# B&R Automation Studio project mvDemoTrak
Automation Studio 4.12.4.107 SP; technology packages: mapp 5.22.1, mappCockpit 5.22.0, mappMotion 5.22.1, mappView 5.22.1

## Configuration CP3686X

### Hardware
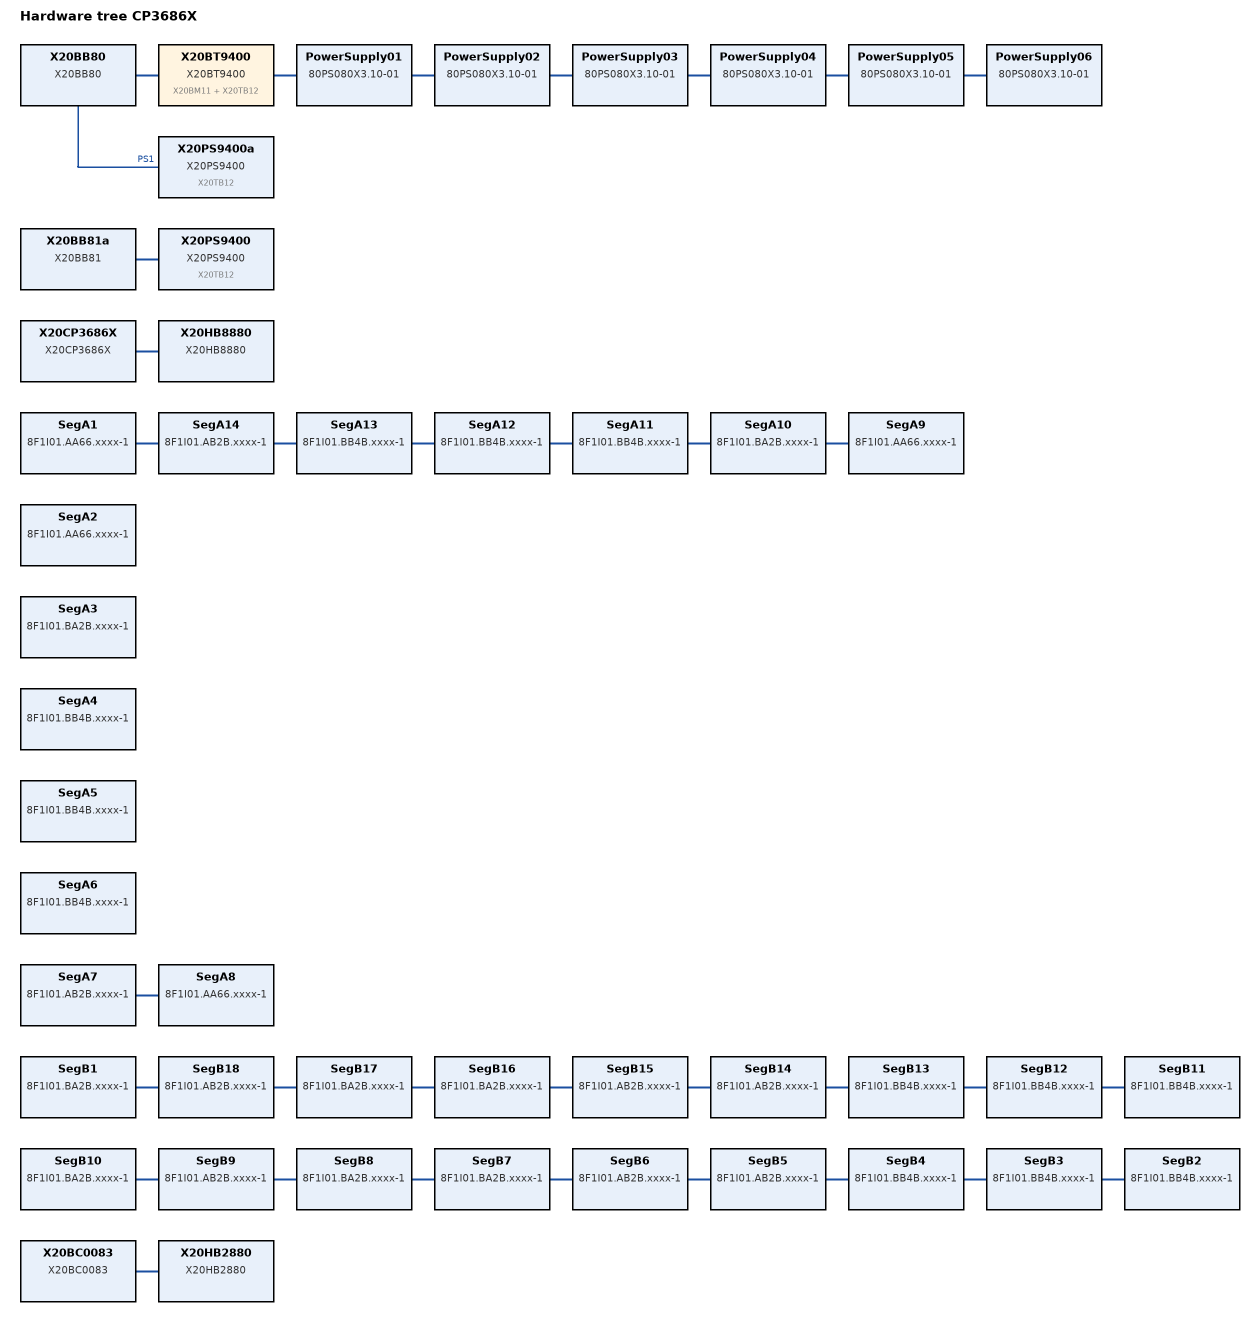
```
PowerSupply01 : 80PS080X3.10-01 v1.5.0.0  [X2X1 -> X20BT9400.X2X1 [Cable Type=X2XCable, Length=10, Version=1.0.0.3]]
  Supervision = off
PowerSupply02 : 80PS080X3.10-01 v1.5.0.0  [X2X1 -> PowerSupply01.X2X2 [Cable Type=X2XCable, Length=10, Version=1.0.0.3]]
  Supervision = off
PowerSupply03 : 80PS080X3.10-01 v1.5.0.0  [X2X1 -> PowerSupply02.X2X2 [Cable Type=X2XCable, Length=10, Version=1.0.0.3]]
  Supervision = off
PowerSupply04 : 80PS080X3.10-01 v1.5.0.0  [X2X1 -> PowerSupply03.X2X2 [Cable Type=X2XCable, Length=10, Version=1.0.0.3]]
  Supervision = off
PowerSupply05 : 80PS080X3.10-01 v1.5.0.0  [X2X1 -> PowerSupply04.X2X2 [Cable Type=X2XCable, Length=10, Version=1.0.0.3]]
  Supervision = off
PowerSupply06 : 80PS080X3.10-01 v1.5.0.0  [X2X1 -> PowerSupply05.X2X2 [Cable Type=X2XCable, Length=10, Version=1.0.0.3]]
  Supervision = off
SegA1 : 8F1I01.AA66.xxxx-1 v1.0.0.2  [PLK1 -> SegA2.PLK2 (NodeNumber=1) [Cable Type=PowerlinkCable, Length=10, Version=1.0.0.3]; PLK2 -> SegA14.PLK1 (NodeNumber=1) [Cable Type=PowerlinkCable, Length=10, Version=1.0.0.3]; PLK3 -> X20HB8880.ETH2 (NodeNumber=1) [Cable Type=PowerlinkCable, Length=10, Version=1.0.0.3]]
  DriveConfiguration:
    McTypeID = LLMConfig
  DriveConfiguration/Segment:
    Shape = STRAIGHT660
    SegmentReference = gSegA1
    SegmentSectorDirection = Positive
    ElongationCompensation = UseAssemblySetting
    StopReaction = UseAssemblySetting
    SpeedFilter = UseAssemblySetting
SegA10 : 8F1I01.BA2B.xxxx-1 v1.0.0.2  [PLK1 -> SegA11.PLK2 (NodeNumber=25) [Cable Type=PowerlinkCable, Length=10, Version=1.0.0.3]; PLK2 -> SegA9.PLK1 (NodeNumber=25) [Cable Type=PowerlinkCable, Length=10, Version=1.0.0.3]]
  DriveConfiguration:
    McTypeID = LLMConfig
  DriveConfiguration/Segment:
    Shape = CIRCULAR_TO_STRAIGHT105
    SegmentReference = gSegA10
    SegmentSectorDirection = Positive
    ElongationCompensation = UseAssemblySetting
    StopReaction = UseAssemblySetting
    SpeedFilter = UseAssemblySetting
SegA11 : 8F1I01.BB4B.xxxx-1 v1.0.0.2  [PLK1 -> SegA12.PLK2 (NodeNumber=24) [Cable Type=PowerlinkCable, Length=10, Version=1.0.0.3]; PLK2 -> SegA10.PLK1 (NodeNumber=24) [Cable Type=PowerlinkCable, Length=10, Version=1.0.0.3]]
  DriveConfiguration:
    McTypeID = LLMConfig
  DriveConfiguration/Segment:
    Shape = CIRCULAR
    SegmentReference = gSegA11
    SegmentSectorDirection = Positive
    ElongationCompensation = UseAssemblySetting
    StopReaction = UseAssemblySetting
    SpeedFilter = UseAssemblySetting
SegA12 : 8F1I01.BB4B.xxxx-1 v1.0.0.2  [PLK1 -> SegA13.PLK2 (NodeNumber=23) [Cable Type=PowerlinkCable, Length=10, Version=1.0.0.3]; PLK2 -> SegA11.PLK1 (NodeNumber=23) [Cable Type=PowerlinkCable, Length=10, Version=1.0.0.3]]
  DriveConfiguration:
    McTypeID = LLMConfig
  DriveConfiguration/Segment:
    Shape = CIRCULAR
    SegmentReference = gSegA12
    SegmentSectorDirection = Positive
    ElongationCompensation = UseAssemblySetting
    StopReaction = UseAssemblySetting
    SpeedFilter = UseAssemblySetting
SegA13 : 8F1I01.BB4B.xxxx-1 v1.0.0.2  [PLK1 -> SegA14.PLK2 (NodeNumber=22) [Cable Type=PowerlinkCable, Length=10, Version=1.0.0.3]; PLK2 -> SegA12.PLK1 (NodeNumber=22) [Cable Type=PowerlinkCable, Length=10, Version=1.0.0.3]]
  DriveConfiguration:
    McTypeID = LLMConfig
  DriveConfiguration/Segment:
    Shape = CIRCULAR
    SegmentReference = gSegA13
    SegmentSectorDirection = Positive
    ElongationCompensation = UseAssemblySetting
    StopReaction = UseAssemblySetting
    SpeedFilter = UseAssemblySetting
SegA14 : 8F1I01.AB2B.xxxx-1 v1.0.0.2  [PLK1 -> SegA1.PLK2 (NodeNumber=21) [Cable Type=PowerlinkCable, Length=10, Version=1.0.0.3]; PLK2 -> SegA13.PLK1 (NodeNumber=21) [Cable Type=PowerlinkCable, Length=10, Version=1.0.0.3]]
  DriveConfiguration:
    McTypeID = LLMConfig
  DriveConfiguration/Segment:
    Shape = STRAIGHT105_TO_CIRCULAR
    SegmentReference = gSegA14
    SegmentSectorDirection = Positive
    ElongationCompensation = UseAssemblySetting
    StopReaction = UseAssemblySetting
    SpeedFilter = UseAssemblySetting
SegA2 : 8F1I01.AA66.xxxx-1 v1.0.0.2  [PLK1 -> SegA3.PLK2 (NodeNumber=2) [Cable Type=PowerlinkCable, Length=10, Version=1.0.0.3]; PLK2 -> SegA1.PLK1 (NodeNumber=2) [Cable Type=PowerlinkCable, Length=10, Version=1.0.0.3]]
  DriveConfiguration:
    McTypeID = LLMConfig
  DriveConfiguration/Segment:
    Shape = STRAIGHT660
    SegmentReference = gSegA2
    SegmentSectorDirection = Positive
    ElongationCompensation = UseAssemblySetting
    StopReaction = UseAssemblySetting
    SpeedFilter = UseAssemblySetting
SegA3 : 8F1I01.BA2B.xxxx-1 v1.0.0.2  [PLK1 -> SegA4.PLK2 (NodeNumber=27) [Cable Type=PowerlinkCable, Length=10, Version=1.0.0.3]; PLK2 -> SegA2.PLK1 (NodeNumber=27) [Cable Type=PowerlinkCable, Length=10, Version=1.0.0.3]]
  DriveConfiguration:
    McTypeID = LLMConfig
  DriveConfiguration/Segment:
    Shape = CIRCULAR_TO_STRAIGHT105
    SegmentReference = gSegA3
    SegmentSectorDirection = Positive
    ElongationCompensation = UseAssemblySetting
    StopReaction = UseAssemblySetting
    SpeedFilter = UseAssemblySetting
SegA4 : 8F1I01.BB4B.xxxx-1 v1.0.0.2  [PLK1 -> SegA5.PLK2 (NodeNumber=28) [Cable Type=PowerlinkCable, Length=10, Version=1.0.0.3]; PLK2 -> SegA3.PLK1 (NodeNumber=28) [Cable Type=PowerlinkCable, Length=10, Version=1.0.0.3]]
  DriveConfiguration:
    McTypeID = LLMConfig
  DriveConfiguration/Segment:
    Shape = CIRCULAR
    SegmentReference = gSegA4
    SegmentSectorDirection = Positive
    ElongationCompensation = UseAssemblySetting
    StopReaction = UseAssemblySetting
    SpeedFilter = UseAssemblySetting
SegA5 : 8F1I01.BB4B.xxxx-1 v1.0.0.2  [PLK1 -> SegA6.PLK2 (NodeNumber=29) [Cable Type=PowerlinkCable, Length=10, Version=1.0.0.3]; PLK2 -> SegA4.PLK1 (NodeNumber=29) [Cable Type=PowerlinkCable, Length=10, Version=1.0.0.3]]
  DriveConfiguration:
    McTypeID = LLMConfig
  DriveConfiguration/Segment:
    Shape = CIRCULAR
    SegmentReference = gSegA5
    SegmentSectorDirection = Positive
    ElongationCompensation = UseAssemblySetting
    StopReaction = UseAssemblySetting
    SpeedFilter = UseAssemblySetting
SegA6 : 8F1I01.BB4B.xxxx-1 v1.0.0.2  [PLK1 -> SegA7.PLK2 (NodeNumber=30) [Cable Type=PowerlinkCable, Length=10, Version=1.0.0.3]; PLK2 -> SegA5.PLK1 (NodeNumber=30) [Cable Type=PowerlinkCable, Length=10, Version=1.0.0.3]]
  DriveConfiguration:
    McTypeID = LLMConfig
  DriveConfiguration/Segment:
    Shape = CIRCULAR
    SegmentReference = gSegA6
    SegmentSectorDirection = Positive
    ElongationCompensation = UseAssemblySetting
    StopReaction = UseAssemblySetting
    SpeedFilter = UseAssemblySetting
SegA7 : 8F1I01.AB2B.xxxx-1 v1.0.0.2  [PLK1 -> SegA8.PLK2 (NodeNumber=31) [Cable Type=PowerlinkCable, Length=10, Version=1.0.0.3]; PLK2 -> SegA6.PLK1 (NodeNumber=31) [Cable Type=PowerlinkCable, Length=10, Version=1.0.0.3]]
  DriveConfiguration:
    McTypeID = LLMConfig
  DriveConfiguration/Segment:
    Shape = STRAIGHT105_TO_CIRCULAR
    SegmentReference = gSegA7
    SegmentSectorDirection = Positive
    ElongationCompensation = UseAssemblySetting
    StopReaction = UseAssemblySetting
    SpeedFilter = UseAssemblySetting
SegA8 : 8F1I01.AA66.xxxx-1 v1.0.0.2  [PLK2 -> SegA7.PLK1 (NodeNumber=32) [Cable Type=PowerlinkCable, Length=10, Version=1.0.0.3]]
  DriveConfiguration:
    McTypeID = LLMConfig
  DriveConfiguration/Segment:
    Shape = STRAIGHT660
    SegmentReference = gSegA8
    SegmentSectorDirection = Positive
    ElongationCompensation = UseAssemblySetting
    StopReaction = UseAssemblySetting
    SpeedFilter = UseAssemblySetting
SegA9 : 8F1I01.AA66.xxxx-1 v1.0.0.2  [PLK1 -> SegA10.PLK2 (NodeNumber=26) [Cable Type=PowerlinkCable, Length=10, Version=1.0.0.3]]
  DriveConfiguration:
    McTypeID = LLMConfig
  DriveConfiguration/Segment:
    Shape = STRAIGHT660
    SegmentReference = gSegA9
    SegmentSectorDirection = Positive
    ElongationCompensation = UseAssemblySetting
    StopReaction = UseAssemblySetting
    SpeedFilter = UseAssemblySetting
SegB1 : 8F1I01.BA2B.xxxx-1 v1.0.0.2  [PLK1 -> SegB2.PLK2 (NodeNumber=3) [Cable Type=PowerlinkCable, Length=10, Version=1.0.0.3]; PLK2 -> SegB18.PLK1 (NodeNumber=3) [Cable Type=PowerlinkCable, Length=10, Version=1.0.0.3]; PLK3 -> X20HB2880.ETH2 (NodeNumber=3) [Cable Type=PowerlinkCable, Length=10, Version=1.0.0.3]]
  DriveConfiguration:
    McTypeID = LLMConfig
  DriveConfiguration/Segment:
    Shape = CIRCULAR_TO_STRAIGHT105
    SegmentReference = gSegB1
    SegmentSectorDirection = Positive
    ElongationCompensation = UseAssemblySetting
    StopReaction = UseAssemblySetting
    SpeedFilter = UseAssemblySetting
SegB10 : 8F1I01.BA2B.xxxx-1 v1.0.0.2  [PLK2 -> SegB9.PLK1 (NodeNumber=12) [Cable Type=PowerlinkCable, Length=10, Version=1.0.0.3]]
  DriveConfiguration:
    McTypeID = LLMConfig
  DriveConfiguration/Segment:
    Shape = CIRCULAR_TO_STRAIGHT105
    SegmentReference = gSegB10
    SegmentSectorDirection = Positive
    ElongationCompensation = UseAssemblySetting
    StopReaction = UseAssemblySetting
    SpeedFilter = UseAssemblySetting
SegB11 : 8F1I01.BB4B.xxxx-1 v1.0.0.2  [PLK1 -> SegB12.PLK2 (NodeNumber=11) [Cable Type=PowerlinkCable, Length=10, Version=1.0.0.3]]
  DriveConfiguration:
    McTypeID = LLMConfig
  DriveConfiguration/Segment:
    Shape = CIRCULAR
    SegmentReference = gSegB11
    SegmentSectorDirection = Positive
    ElongationCompensation = UseAssemblySetting
    StopReaction = UseAssemblySetting
    SpeedFilter = UseAssemblySetting
SegB12 : 8F1I01.BB4B.xxxx-1 v1.0.0.2  [PLK1 -> SegB13.PLK2 (NodeNumber=10) [Cable Type=PowerlinkCable, Length=10, Version=1.0.0.3]; PLK2 -> SegB11.PLK1 (NodeNumber=10) [Cable Type=PowerlinkCable, Length=10, Version=1.0.0.3]]
  DriveConfiguration:
    McTypeID = LLMConfig
  DriveConfiguration/Segment:
    Shape = CIRCULAR
    SegmentReference = gSegB12
    SegmentSectorDirection = Positive
    ElongationCompensation = UseAssemblySetting
    StopReaction = UseAssemblySetting
    SpeedFilter = UseAssemblySetting
SegB13 : 8F1I01.BB4B.xxxx-1 v1.0.0.2  [PLK1 -> SegB14.PLK2 (NodeNumber=9) [Cable Type=PowerlinkCable, Length=10, Version=1.0.0.3]; PLK2 -> SegB12.PLK1 (NodeNumber=9) [Cable Type=PowerlinkCable, Length=10, Version=1.0.0.3]]
  DriveConfiguration:
    McTypeID = LLMConfig
  DriveConfiguration/Segment:
    Shape = CIRCULAR
    SegmentReference = gSegB13
    SegmentSectorDirection = Positive
    ElongationCompensation = UseAssemblySetting
    StopReaction = UseAssemblySetting
    SpeedFilter = UseAssemblySetting
SegB14 : 8F1I01.AB2B.xxxx-1 v1.0.0.2  [PLK1 -> SegB15.PLK2 (NodeNumber=8) [Cable Type=PowerlinkCable, Length=10, Version=1.0.0.3]; PLK2 -> SegB13.PLK1 (NodeNumber=8) [Cable Type=PowerlinkCable, Length=10, Version=1.0.0.3]]
  DriveConfiguration:
    McTypeID = LLMConfig
  DriveConfiguration/Segment:
    Shape = STRAIGHT105_TO_CIRCULAR
    SegmentReference = gSegB14
    SegmentSectorDirection = Positive
    ElongationCompensation = UseAssemblySetting
    StopReaction = UseAssemblySetting
    SpeedFilter = UseAssemblySetting
SegB15 : 8F1I01.AB2B.xxxx-1 v1.0.0.2  [PLK1 -> SegB16.PLK2 (NodeNumber=7) [Cable Type=PowerlinkCable, Length=10, Version=1.0.0.3]; PLK2 -> SegB14.PLK1 (NodeNumber=7) [Cable Type=PowerlinkCable, Length=10, Version=1.0.0.3]]
  DriveConfiguration:
    McTypeID = LLMConfig
  DriveConfiguration/Segment:
    Shape = STRAIGHT105_TO_CIRCULAR
    SegmentReference = gSegB15
    SegmentSectorDirection = Positive
    ElongationCompensation = UseAssemblySetting
    StopReaction = UseAssemblySetting
    SpeedFilter = UseAssemblySetting
SegB16 : 8F1I01.BA2B.xxxx-1 v1.0.0.2  [PLK1 -> SegB17.PLK2 (NodeNumber=6) [Cable Type=PowerlinkCable, Length=10, Version=1.0.0.3]; PLK2 -> SegB15.PLK1 (NodeNumber=6) [Cable Type=PowerlinkCable, Length=10, Version=1.0.0.3]]
  DriveConfiguration:
    McTypeID = LLMConfig
  DriveConfiguration/Segment:
    Shape = CIRCULAR_TO_STRAIGHT105
    SegmentReference = gSegB16
    SegmentSectorDirection = Positive
    ElongationCompensation = UseAssemblySetting
    StopReaction = UseAssemblySetting
    SpeedFilter = UseAssemblySetting
SegB17 : 8F1I01.BA2B.xxxx-1 v1.0.0.2  [PLK1 -> SegB18.PLK2 (NodeNumber=5) [Cable Type=PowerlinkCable, Length=10, Version=1.0.0.3]; PLK2 -> SegB16.PLK1 (NodeNumber=5) [Cable Type=PowerlinkCable, Length=10, Version=1.0.0.3]]
  DriveConfiguration:
    McTypeID = LLMConfig
  DriveConfiguration/Segment:
    Shape = CIRCULAR_TO_STRAIGHT105
    SegmentReference = gSegB17
    SegmentSectorDirection = Positive
    ElongationCompensation = UseAssemblySetting
    StopReaction = UseAssemblySetting
    SpeedFilter = UseAssemblySetting
SegB18 : 8F1I01.AB2B.xxxx-1 v1.0.0.2  [PLK1 -> SegB1.PLK2 (NodeNumber=4) [Cable Type=PowerlinkCable, Length=10, Version=1.0.0.3]; PLK2 -> SegB17.PLK1 (NodeNumber=4) [Cable Type=PowerlinkCable, Length=10, Version=1.0.0.3]]
  DriveConfiguration:
    McTypeID = LLMConfig
  DriveConfiguration/Segment:
    Shape = STRAIGHT105_TO_CIRCULAR
    SegmentReference = gSegB18
    SegmentSectorDirection = Positive
    ElongationCompensation = UseAssemblySetting
    StopReaction = UseAssemblySetting
    SpeedFilter = UseAssemblySetting
SegB2 : 8F1I01.BB4B.xxxx-1 v1.0.0.2  [PLK1 -> SegB3.PLK2 (NodeNumber=13) [Cable Type=PowerlinkCable, Length=10, Version=1.0.0.3]; PLK2 -> SegB1.PLK1 (NodeNumber=13) [Cable Type=PowerlinkCable, Length=10, Version=1.0.0.3]]
  DriveConfiguration:
    McTypeID = LLMConfig
  DriveConfiguration/Segment:
    Shape = CIRCULAR
    SegmentReference = gSegB2
    SegmentSectorDirection = Positive
    ElongationCompensation = UseAssemblySetting
    StopReaction = UseAssemblySetting
    SpeedFilter = UseAssemblySetting
SegB3 : 8F1I01.BB4B.xxxx-1 v1.0.0.2  [PLK1 -> SegB4.PLK2 (NodeNumber=14) [Cable Type=PowerlinkCable, Length=10, Version=1.0.0.3]; PLK2 -> SegB2.PLK1 (NodeNumber=14) [Cable Type=PowerlinkCable, Length=10, Version=1.0.0.3]]
  DriveConfiguration:
    McTypeID = LLMConfig
  DriveConfiguration/Segment:
    Shape = CIRCULAR
    SegmentReference = gSegB3
    SegmentSectorDirection = Positive
    ElongationCompensation = UseAssemblySetting
    StopReaction = UseAssemblySetting
    SpeedFilter = UseAssemblySetting
SegB4 : 8F1I01.BB4B.xxxx-1 v1.0.0.2  [PLK1 -> SegB5.PLK2 (NodeNumber=15) [Cable Type=PowerlinkCable, Length=10, Version=1.0.0.3]; PLK2 -> SegB3.PLK1 (NodeNumber=15) [Cable Type=PowerlinkCable, Length=10, Version=1.0.0.3]]
  DriveConfiguration:
    McTypeID = LLMConfig
  DriveConfiguration/Segment:
    Shape = CIRCULAR
    SegmentReference = gSegB4
    SegmentSectorDirection = Positive
    ElongationCompensation = UseAssemblySetting
    StopReaction = UseAssemblySetting
    SpeedFilter = UseAssemblySetting
SegB5 : 8F1I01.AB2B.xxxx-1 v1.0.0.2  [PLK1 -> SegB6.PLK2 (NodeNumber=16) [Cable Type=PowerlinkCable, Length=10, Version=1.0.0.3]; PLK2 -> SegB4.PLK1 (NodeNumber=16) [Cable Type=PowerlinkCable, Length=10, Version=1.0.0.3]]
  DriveConfiguration:
    McTypeID = LLMConfig
  DriveConfiguration/Segment:
    Shape = STRAIGHT105_TO_CIRCULAR
    SegmentReference = gSegB5
    SegmentSectorDirection = Positive
    ElongationCompensation = UseAssemblySetting
    StopReaction = UseAssemblySetting
    SpeedFilter = UseAssemblySetting
SegB6 : 8F1I01.AB2B.xxxx-1 v1.0.0.2  [PLK1 -> SegB7.PLK2 (NodeNumber=17) [Cable Type=PowerlinkCable, Length=10, Version=1.0.0.3]; PLK2 -> SegB5.PLK1 (NodeNumber=17) [Cable Type=PowerlinkCable, Length=10, Version=1.0.0.3]]
  DriveConfiguration:
    McTypeID = LLMConfig
  DriveConfiguration/Segment:
    Shape = STRAIGHT105_TO_CIRCULAR
    SegmentReference = gSegB6
    SegmentSectorDirection = Positive
    ElongationCompensation = UseAssemblySetting
    StopReaction = UseAssemblySetting
    SpeedFilter = UseAssemblySetting
SegB7 : 8F1I01.BA2B.xxxx-1 v1.0.0.2  [PLK1 -> SegB8.PLK2 (NodeNumber=18) [Cable Type=PowerlinkCable, Length=10, Version=1.0.0.3]; PLK2 -> SegB6.PLK1 (NodeNumber=18) [Cable Type=PowerlinkCable, Length=10, Version=1.0.0.3]]
  DriveConfiguration:
    McTypeID = LLMConfig
  DriveConfiguration/Segment:
    Shape = CIRCULAR_TO_STRAIGHT105
    SegmentReference = gSegB7
    SegmentSectorDirection = Positive
    ElongationCompensation = UseAssemblySetting
    StopReaction = UseAssemblySetting
    SpeedFilter = UseAssemblySetting
SegB8 : 8F1I01.BA2B.xxxx-1 v1.0.0.2  [PLK1 -> SegB9.PLK2 (NodeNumber=20) [Cable Type=PowerlinkCable, Length=10, Version=1.0.0.3]; PLK2 -> SegB7.PLK1 (NodeNumber=20) [Cable Type=PowerlinkCable, Length=10, Version=1.0.0.3]]
  DriveConfiguration:
    McTypeID = LLMConfig
  DriveConfiguration/Segment:
    Shape = CIRCULAR_TO_STRAIGHT105
    SegmentReference = gSegB8
    SegmentSectorDirection = Positive
    ElongationCompensation = UseAssemblySetting
    StopReaction = UseAssemblySetting
    SpeedFilter = UseAssemblySetting
SegB9 : 8F1I01.AB2B.xxxx-1 v1.0.0.2  [PLK1 -> SegB10.PLK2 (NodeNumber=19) [Cable Type=PowerlinkCable, Length=10, Version=1.0.0.3]; PLK2 -> SegB8.PLK1 (NodeNumber=19) [Cable Type=PowerlinkCable, Length=10, Version=1.0.0.3]]
  DriveConfiguration:
    McTypeID = LLMConfig
  DriveConfiguration/Segment:
    Shape = STRAIGHT105_TO_CIRCULAR
    SegmentReference = gSegB9
    SegmentSectorDirection = Positive
    ElongationCompensation = UseAssemblySetting
    StopReaction = UseAssemblySetting
    SpeedFilter = UseAssemblySetting
X20BB80 : X20BB80 v1.1.0.0
X20BB81a : X20BB81 v1.1.0.0
  Connector IF1:
    ActivateX2X = 0
X20BC0083 : X20BC0083 v2.14.0.0  [PLK1 -> X20HB2880.ETH1 (NodeNumber=33) [Cable Type=PowerlinkCable, Length=10, Version=1.0.0.3]; SL -> X20BB80.SL1]
  Supervision = off
X20BM11 : X20BM11 v1.1.0.0  [X2X1 -> X20BB80.IF1]
X20BT9400 : X20BT9400 v1.3.0.0  [SS1 -> X20TB12b.SS; SL -> X20BM11.SL1]
  Supervision = off
X20CP3686X : X20CP3686X v1.6.2.0
  Connector IF2:
    ActivateDevice = 1
    Mode = Manual
    InternetAddress = 192.168.0.105
    SubnetMask = 255.255.255.0
    ActivateSnmp = 2
  Connector IF3:
    CycleTime = 2000
  ConfigurationID = mvDemoTrak_CP1685
  ConfigVersion = 1.1.0
  MotionLoggerSize = 2048000
  EnableUsbRemoteInstall = 1
  TimerDeviceType = EPLX2X
  TimerDevice = X20CP3686X.IF3
  TaskClassIdleTime = 2000
  Cyclic1Duration = 2000
  Cyclic1Tolerance = 0
  Cyclic2Duration = 10000
  Cyclic2Tolerance = 10000
  FileDevice1
  FileDeviceName1 = SvgData
  FileDevicePath1 = USER_PATH\web\SvgData
  FileDevice2
  FileDeviceName2 = Diagnosis
  FileDevicePath2 = USER_PATH\web\Diagnosis
  FileDevice3
  FileDeviceName3 = USER
  FileDevicePath3 = USER_PATH\
  FtpUser1
  FtpUsername1 = Admin
  FtpUserPassword1 = b2dkeklN0DR4HlzomfG8N5dlVtI3Hrgd5HBjTL6T4A4=  // pw: admin
  FtpUserSalt1 = LZ6GLOae
  FTPAccessRight1 = 0
  FTPdevice1 = ALL
  FtpUser2
  FtpUsername2 = service
  FtpUserPassword2 = y0+bdtT85NEfd+yInx4lMGxqzvQGY/+IGfzWbkQcI6M=
  FtpUserSalt2 = 0i04Zj6L
  FTPAccessRight2 = 0
  FTPMSpath2 = web\Diagnosis
  WebServerWebDir = USER_PATH\web  // default: web\
  ActivateOpcUa = 1
  OpcUaInformationModels_PV_Version = 1
X20HB2880 : X20HB2880 v1.2.0.0  [ETH1 -> X20BC0083.PLK1 [Cable Type=PowerlinkCable, Length=10, Version=1.0.0.3]; ETH2 -> SegB1.PLK3 [Cable Type=PowerlinkCable, Length=10, Version=1.0.0.3]; SS -> X20BB81a.SS1]
X20HB8880 : X20HB8880 v1.1.0.0  [ETH1 -> X20CP3686X.IF3 [Cable Type=PowerlinkCable, Length=10, Version=1.0.0.3]; ETH2 -> SegA1.PLK3 [Cable Type=PowerlinkCable, Length=10, Version=1.0.0.3]; SL -> X20BB81a.SL1]
X20PS9400 : X20PS9400 v1.8.0.0  [SS1 -> X20TB12.SS; PS -> X20BB81a.PS1]
  Supervision = off
X20PS9400a : X20PS9400 v1.8.0.0  [SS1 -> X20TB12a.SS; PS -> X20BB80.PS1]
  Supervision = off
X20TB12 : X20TB12 v1.0.0.0
X20TB12a : X20TB12 v1.0.0.0
X20TB12b : X20TB12 v1.0.0.0
```

## Configuration Config1

CPU 5PC900.TS17-00, AutomationRuntime D4.93, Build 6.3.0, Safety 0.0, Vc 

### Task classes (Cpu.sw)
```
Cyclic#1 (cycle 2000 us, tolerance 0 us):
  TrakInit <- Trak.TrakInit.prg
Cyclic#2 (cycle 10000 us, tolerance 10000 us):
  AssCtrl <- Trak.AssCtrl.prg
  AlarmXTask <- VisuPackage.AlarmXTask.prg
  VisuTask <- VisuPackage.VisuTask.prg
Cyclic#4:
  SegCtrl <- Trak.SegCtrl.prg
Cyclic#8:
  FileExplor <- mappFileExplorer.FileExplorer.prg
  UsbDevice <- USBdevice.UsbDevice.prg
  NetDevice <- NETdevice.NetDevice.prg
DataObjects: McAcpSys
NcDataObjects: mcdrivelog
Binaries: McAcpSim, FWRules, arcoal, arsvcreg, TCData, McAcpDrv, mCoWebSc, mvLoader, arflatprv, udbdef, TCLang, iomap, Config_1, arconfig, asfw, ashwac, sysconf, User, Settings, Role, ashwd, Config_4, Config_3, Config_2, Config, CfgAlHist, TC, CfgAlList
Libraries: McBase, CoTrace, AsZip, FileIO, runtime, McAxis, McAcpTrak, MpBase, TrakLib, standard, AsBrStr, sys_lib, brsystem, astime, ArEventLog, DataObj, AsHttp, MpServer, TrakDiag, AsArSdm, MpAlarmX, AsMem, AsUSB, powerlnk, arssl, asieccon, aruser, AsICMP
```

### Hardware
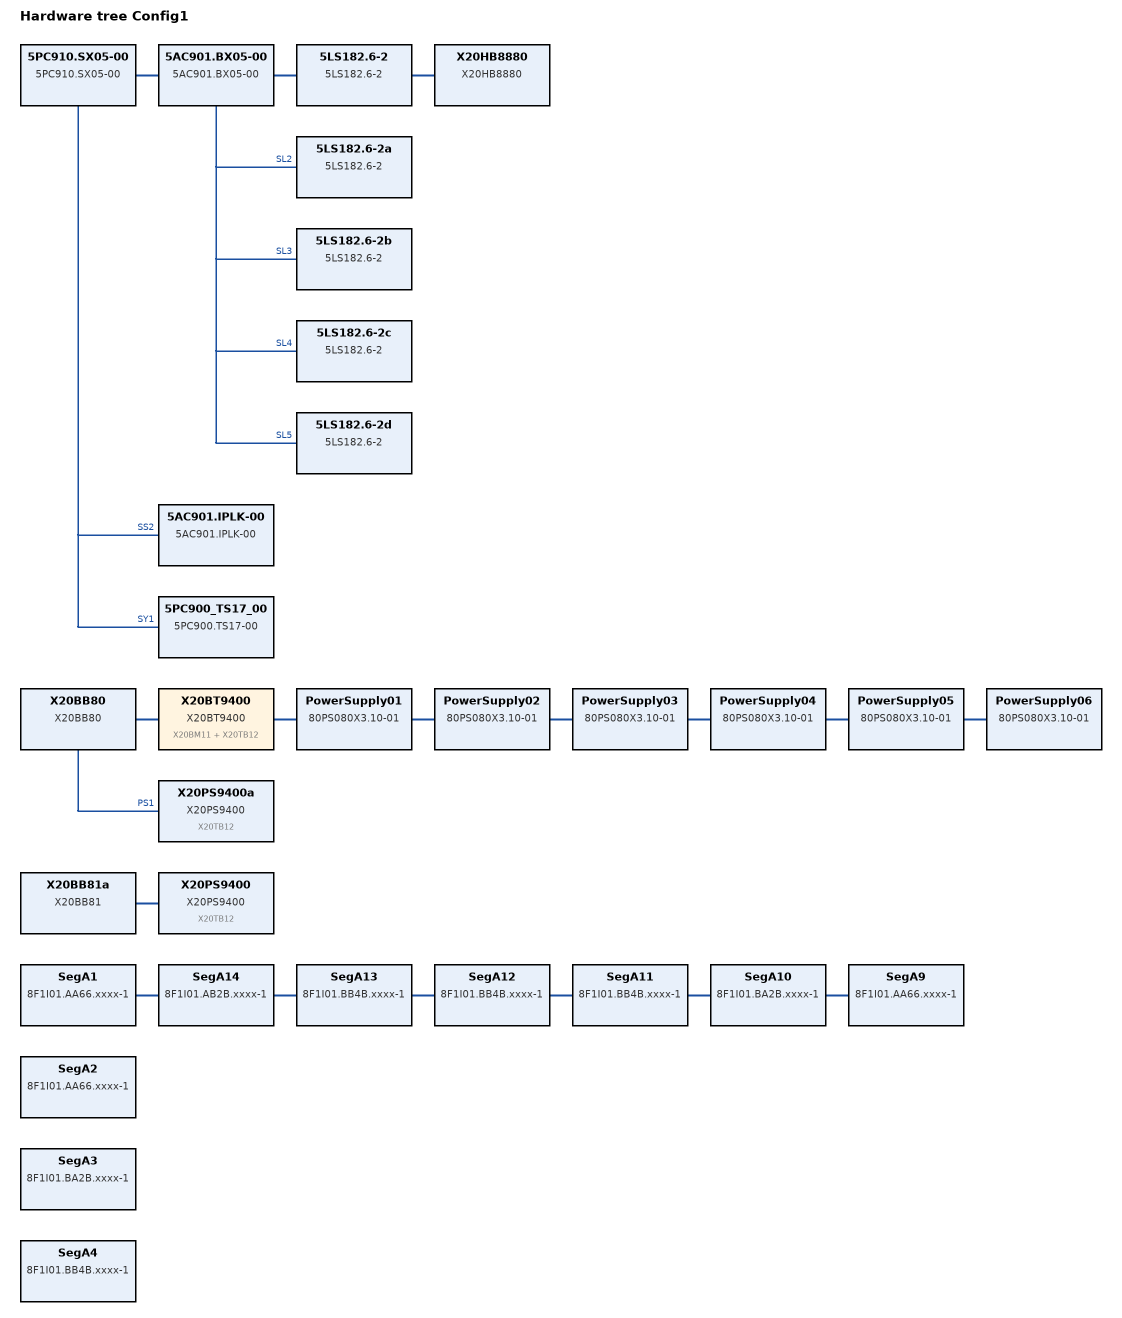
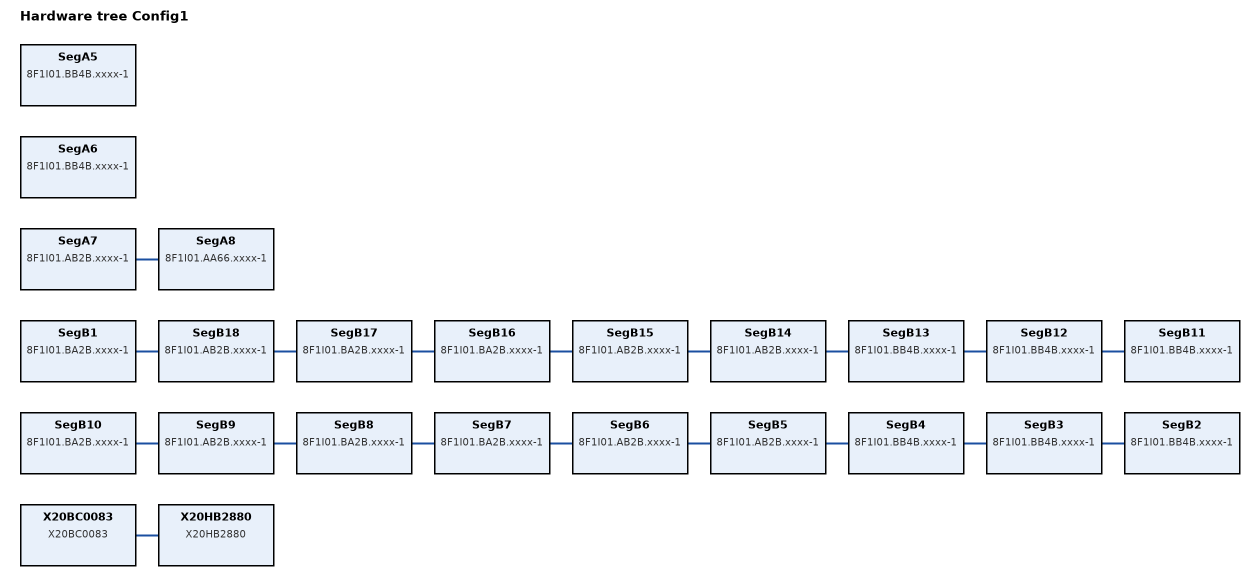
```
5AC901.BX05-00 : 5AC901.BX05-00 v1.0.1.0  [SY -> 5PC910.SX05-00.SY3]
5AC901.IPLK-00 : 5AC901.IPLK-00 v1.8.0.1 (Disabled=true)  [SS -> 5PC910.SX05-00.SS2]
  Connector IF1 (Disabled=true)
5LS182.6-2 : 5LS182.6-2 v1.9.0.0  [SL -> 5AC901.BX05-00.SL1]
  Connector IF1:
    EplHostName = mvdemotrak
    NodeDefinition = Software
    HostName = mvdemotrak
5LS182.6-2a : 5LS182.6-2 v1.9.0.0 (Disabled=true)  [SL -> 5AC901.BX05-00.SL2]
  Connector IF1 (Disabled=true)
    EplHostName = mvdemotrak
    HostName = mvdemotrak
5LS182.6-2b : 5LS182.6-2 v1.9.0.0 (Disabled=true)  [SL -> 5AC901.BX05-00.SL3]
  Connector IF1 (Disabled=true)
    EplHostName = mvdemotrak
    HostName = mvdemotrak
5LS182.6-2c : 5LS182.6-2 v1.9.0.0 (Disabled=true)  [SL -> 5AC901.BX05-00.SL4]
  Connector IF1 (Disabled=true)
    EplHostName = mvdemotrak
    HostName = mvdemotrak
5LS182.6-2d : 5LS182.6-2 v1.9.0.0 (Disabled=true)  [SL -> 5AC901.BX05-00.SL5]
  Connector IF1 (Disabled=true)
    EplHostName = mvdemotrak
    HostName = mvdemotrak
5PC900_TS17_00 : 5PC900.TS17-00 v2.1.0.0  [SY -> 5PC910.SX05-00.SY1]
  ConfigurationID = TrakDemo_Config1
  ConfigVersion = 1.2.4
  Simulation = 1
  MotionLoggerSize = 2048000
  TaskClassIdleTime = 3000
  Cyclic1Duration = 2000
  Cyclic1Tolerance = 0
  Cyclic2Duration = 10000
  Cyclic2Tolerance = 10000
  FileDevice1
  FileDeviceName1 = SvgData
  FileDevicePath1 = USER_PATH\web\SvgData
  FileDevice2
  FileDeviceName2 = Diagnosis
  FileDevicePath2 = USER_PATH\web\Diagnosis
  FileDevice3
  FileDeviceName3 = USER
  FileDevicePath3 = USER_PATH\
  EthernetHostName = mvdemotrak
  EthernetDefaultGateway = 10.49.40.1
  FtpUser1
  FtpUsername1 = admin
  FtpUserPassword1 = 1eFk4bv95gGd/YhutE0/XT32p+eqiGHSQm0YwzXwS3M=
  FtpUserSalt1 = in5n/jXa
  FTPAccessRight1 = 0
  FTPdevice1 = ALL
  FtpUser2
  FtpUsername2 = service
  FtpUserPassword2 = O8ov+IySxWdP6BEBN2hJQHEc5z1frphrSNyvJ0Di8wc=
  FtpUserSalt2 = r1F4c1QQ
  FTPAccessRight2 = 0
  FTPMSpath2 = web\Diagnosis
  WebServerWebDir = USER_PATH\web\
  ActivateOpcUa = 1
  OpcUaInformationModels_PV_Version = 1
5PC910.SX05-00 : 5PC910.SX05-00 v2.1.0.0
  Connector IF1:
    AssignedOperatingSystem = ARemb
  Connector IF3:
    AssignedOperatingSystem = ARemb
    ActivateDevice = 1
    HostName = mvdemotrak
    Mode = Manual
    InternetAddress = 10.49.40.236
    SubnetMask = 255.255.255.0
    ActivateSnmp = 2
  Connector IF4:
    AssignedOperatingSystem = ARemb
    ActivateDevice = 1
    HostName = mvdemotrak
    Mode = Manual
    InternetAddress = 172.16.0.100
    SubnetMask = 255.255.255.0
    ActivateIna = 0
  Connector IF5:
    AssignedOperatingSystem = ARemb
  Connector IF6:
    AssignedOperatingSystem = ARemb
  Connector IF7:
    AssignedOperatingSystem = ARemb
  Connector IF8:
    AssignedOperatingSystem = ARemb
  Connector IF9:
    AssignedOperatingSystem = ARemb
PowerSupply01 : 80PS080X3.10-01 v1.5.0.0  [X2X1 -> X20BT9400.X2X1 [Cable Type=X2XCable, Length=10, Version=1.0.0.3]]
  Supervision = off
PowerSupply02 : 80PS080X3.10-01 v1.5.0.0  [X2X1 -> PowerSupply01.X2X2 [Cable Type=X2XCable, Length=10, Version=1.0.0.3]]
  Supervision = off
PowerSupply03 : 80PS080X3.10-01 v1.5.0.0  [X2X1 -> PowerSupply02.X2X2 [Cable Type=X2XCable, Length=10, Version=1.0.0.3]]
  Supervision = off
PowerSupply04 : 80PS080X3.10-01 v1.5.0.0  [X2X1 -> PowerSupply03.X2X2 [Cable Type=X2XCable, Length=10, Version=1.0.0.3]]
  Supervision = off
PowerSupply05 : 80PS080X3.10-01 v1.5.0.0  [X2X1 -> PowerSupply04.X2X2 [Cable Type=X2XCable, Length=10, Version=1.0.0.3]]
  Supervision = off
PowerSupply06 : 80PS080X3.10-01 v1.5.0.0  [X2X1 -> PowerSupply05.X2X2 [Cable Type=X2XCable, Length=10, Version=1.0.0.3]]
  Supervision = off
SegA1 : 8F1I01.AA66.xxxx-1 v1.0.0.2  [PLK1 -> SegA2.PLK2 (NodeNumber=1) [Cable Type=PowerlinkCable, Length=10, Version=1.0.0.3]; PLK2 -> SegA14.PLK1 (NodeNumber=1) [Cable Type=PowerlinkCable, Length=10, Version=1.0.0.3]; PLK3 -> X20HB8880.ETH2 (NodeNumber=1) [Cable Type=PowerlinkCable, Length=10, Version=1.0.0.3]]
  DriveConfiguration:
    McTypeID = LLMConfig
  DriveConfiguration/Segment:
    Shape = STRAIGHT660
    SegmentReference = gSegA1
    SegmentSectorDirection = Positive
    ElongationCompensation = UseAssemblySetting
    StopReaction = UseAssemblySetting
    SpeedFilter = UseAssemblySetting
SegA10 : 8F1I01.BA2B.xxxx-1 v1.0.0.2  [PLK1 -> SegA11.PLK2 (NodeNumber=25) [Cable Type=PowerlinkCable, Length=10, Version=1.0.0.3]; PLK2 -> SegA9.PLK1 (NodeNumber=25) [Cable Type=PowerlinkCable, Length=10, Version=1.0.0.3]]
  DriveConfiguration:
    McTypeID = LLMConfig
  DriveConfiguration/Segment:
    Shape = CIRCULAR_TO_STRAIGHT105
    SegmentReference = gSegA10
    SegmentSectorDirection = Positive
    ElongationCompensation = UseAssemblySetting
    StopReaction = UseAssemblySetting
    SpeedFilter = UseAssemblySetting
SegA11 : 8F1I01.BB4B.xxxx-1 v1.0.0.2  [PLK1 -> SegA12.PLK2 (NodeNumber=24) [Cable Type=PowerlinkCable, Length=10, Version=1.0.0.3]; PLK2 -> SegA10.PLK1 (NodeNumber=24) [Cable Type=PowerlinkCable, Length=10, Version=1.0.0.3]]
  DriveConfiguration:
    McTypeID = LLMConfig
  DriveConfiguration/Segment:
    Shape = CIRCULAR
    SegmentReference = gSegA11
    SegmentSectorDirection = Positive
    ElongationCompensation = UseAssemblySetting
    StopReaction = UseAssemblySetting
    SpeedFilter = UseAssemblySetting
SegA12 : 8F1I01.BB4B.xxxx-1 v1.0.0.2  [PLK1 -> SegA13.PLK2 (NodeNumber=23) [Cable Type=PowerlinkCable, Length=10, Version=1.0.0.3]; PLK2 -> SegA11.PLK1 (NodeNumber=23) [Cable Type=PowerlinkCable, Length=10, Version=1.0.0.3]]
  DriveConfiguration:
    McTypeID = LLMConfig
  DriveConfiguration/Segment:
    Shape = CIRCULAR
    SegmentReference = gSegA12
    SegmentSectorDirection = Positive
    ElongationCompensation = UseAssemblySetting
    StopReaction = UseAssemblySetting
    SpeedFilter = UseAssemblySetting
SegA13 : 8F1I01.BB4B.xxxx-1 v1.0.0.2  [PLK1 -> SegA14.PLK2 (NodeNumber=22) [Cable Type=PowerlinkCable, Length=10, Version=1.0.0.3]; PLK2 -> SegA12.PLK1 (NodeNumber=22) [Cable Type=PowerlinkCable, Length=10, Version=1.0.0.3]]
  DriveConfiguration:
    McTypeID = LLMConfig
  DriveConfiguration/Segment:
    Shape = CIRCULAR
    SegmentReference = gSegA13
    SegmentSectorDirection = Positive
    ElongationCompensation = UseAssemblySetting
    StopReaction = UseAssemblySetting
    SpeedFilter = UseAssemblySetting
SegA14 : 8F1I01.AB2B.xxxx-1 v1.0.0.2  [PLK1 -> SegA1.PLK2 (NodeNumber=21) [Cable Type=PowerlinkCable, Length=10, Version=1.0.0.3]; PLK2 -> SegA13.PLK1 (NodeNumber=21) [Cable Type=PowerlinkCable, Length=10, Version=1.0.0.3]]
  DriveConfiguration:
    McTypeID = LLMConfig
  DriveConfiguration/Segment:
    Shape = STRAIGHT105_TO_CIRCULAR
    SegmentReference = gSegA14
    SegmentSectorDirection = Positive
    ElongationCompensation = UseAssemblySetting
    StopReaction = UseAssemblySetting
    SpeedFilter = UseAssemblySetting
SegA2 : 8F1I01.AA66.xxxx-1 v1.0.0.2  [PLK1 -> SegA3.PLK2 (NodeNumber=2) [Cable Type=PowerlinkCable, Length=10, Version=1.0.0.3]; PLK2 -> SegA1.PLK1 (NodeNumber=2) [Cable Type=PowerlinkCable, Length=10, Version=1.0.0.3]]
  DriveConfiguration:
    McTypeID = LLMConfig
  DriveConfiguration/Segment:
    Shape = STRAIGHT660
    SegmentReference = gSegA2
    SegmentSectorDirection = Positive
    ElongationCompensation = UseAssemblySetting
    StopReaction = UseAssemblySetting
    SpeedFilter = UseAssemblySetting
SegA3 : 8F1I01.BA2B.xxxx-1 v1.0.0.2  [PLK1 -> SegA4.PLK2 (NodeNumber=27) [Cable Type=PowerlinkCable, Length=10, Version=1.0.0.3]; PLK2 -> SegA2.PLK1 (NodeNumber=27) [Cable Type=PowerlinkCable, Length=10, Version=1.0.0.3]]
  DriveConfiguration:
    McTypeID = LLMConfig
  DriveConfiguration/Segment:
    Shape = CIRCULAR_TO_STRAIGHT105
    SegmentReference = gSegA3
    SegmentSectorDirection = Positive
    ElongationCompensation = UseAssemblySetting
    StopReaction = UseAssemblySetting
    SpeedFilter = UseAssemblySetting
SegA4 : 8F1I01.BB4B.xxxx-1 v1.0.0.2  [PLK1 -> SegA5.PLK2 (NodeNumber=28) [Cable Type=PowerlinkCable, Length=10, Version=1.0.0.3]; PLK2 -> SegA3.PLK1 (NodeNumber=28) [Cable Type=PowerlinkCable, Length=10, Version=1.0.0.3]]
  DriveConfiguration:
    McTypeID = LLMConfig
  DriveConfiguration/Segment:
    Shape = CIRCULAR
    SegmentReference = gSegA4
    SegmentSectorDirection = Positive
    ElongationCompensation = UseAssemblySetting
    StopReaction = UseAssemblySetting
    SpeedFilter = UseAssemblySetting
SegA5 : 8F1I01.BB4B.xxxx-1 v1.0.0.2  [PLK1 -> SegA6.PLK2 (NodeNumber=29) [Cable Type=PowerlinkCable, Length=10, Version=1.0.0.3]; PLK2 -> SegA4.PLK1 (NodeNumber=29) [Cable Type=PowerlinkCable, Length=10, Version=1.0.0.3]]
  DriveConfiguration:
    McTypeID = LLMConfig
  DriveConfiguration/Segment:
    Shape = CIRCULAR
    SegmentReference = gSegA5
    SegmentSectorDirection = Positive
    ElongationCompensation = UseAssemblySetting
    StopReaction = UseAssemblySetting
    SpeedFilter = UseAssemblySetting
SegA6 : 8F1I01.BB4B.xxxx-1 v1.0.0.2  [PLK1 -> SegA7.PLK2 (NodeNumber=30) [Cable Type=PowerlinkCable, Length=10, Version=1.0.0.3]; PLK2 -> SegA5.PLK1 (NodeNumber=30) [Cable Type=PowerlinkCable, Length=10, Version=1.0.0.3]]
  DriveConfiguration:
    McTypeID = LLMConfig
  DriveConfiguration/Segment:
    Shape = CIRCULAR
    SegmentReference = gSegA6
    SegmentSectorDirection = Positive
    ElongationCompensation = UseAssemblySetting
    StopReaction = UseAssemblySetting
    SpeedFilter = UseAssemblySetting
SegA7 : 8F1I01.AB2B.xxxx-1 v1.0.0.2  [PLK1 -> SegA8.PLK2 (NodeNumber=31) [Cable Type=PowerlinkCable, Length=10, Version=1.0.0.3]; PLK2 -> SegA6.PLK1 (NodeNumber=31) [Cable Type=PowerlinkCable, Length=10, Version=1.0.0.3]]
  DriveConfiguration:
    McTypeID = LLMConfig
  DriveConfiguration/Segment:
    Shape = STRAIGHT105_TO_CIRCULAR
    SegmentReference = gSegA7
    SegmentSectorDirection = Positive
    ElongationCompensation = UseAssemblySetting
    StopReaction = UseAssemblySetting
    SpeedFilter = UseAssemblySetting
SegA8 : 8F1I01.AA66.xxxx-1 v1.0.0.2  [PLK2 -> SegA7.PLK1 (NodeNumber=32) [Cable Type=PowerlinkCable, Length=10, Version=1.0.0.3]]
  DriveConfiguration:
    McTypeID = LLMConfig
  DriveConfiguration/Segment:
    Shape = STRAIGHT660
    SegmentReference = gSegA8
    SegmentSectorDirection = Positive
    ElongationCompensation = UseAssemblySetting
    StopReaction = UseAssemblySetting
    SpeedFilter = UseAssemblySetting
SegA9 : 8F1I01.AA66.xxxx-1 v1.0.0.2  [PLK1 -> SegA10.PLK2 (NodeNumber=26) [Cable Type=PowerlinkCable, Length=10, Version=1.0.0.3]]
  DriveConfiguration:
    McTypeID = LLMConfig
  DriveConfiguration/Segment:
    Shape = STRAIGHT660
    SegmentReference = gSegA9
    SegmentSectorDirection = Positive
    ElongationCompensation = UseAssemblySetting
    StopReaction = UseAssemblySetting
    SpeedFilter = UseAssemblySetting
SegB1 : 8F1I01.BA2B.xxxx-1 v1.0.0.2  [PLK1 -> SegB2.PLK2 (NodeNumber=3) [Cable Type=PowerlinkCable, Length=10, Version=1.0.0.3]; PLK2 -> SegB18.PLK1 (NodeNumber=3) [Cable Type=PowerlinkCable, Length=10, Version=1.0.0.3]; PLK3 -> X20HB2880.ETH2 (NodeNumber=3) [Cable Type=PowerlinkCable, Length=10, Version=1.0.0.3]]
  DriveConfiguration:
    McTypeID = LLMConfig
  DriveConfiguration/Segment:
    Shape = CIRCULAR_TO_STRAIGHT105
    SegmentReference = gSegB1
    SegmentSectorDirection = Positive
    ElongationCompensation = UseAssemblySetting
    StopReaction = UseAssemblySetting
    SpeedFilter = UseAssemblySetting
SegB10 : 8F1I01.BA2B.xxxx-1 v1.0.0.2  [PLK2 -> SegB9.PLK1 (NodeNumber=12) [Cable Type=PowerlinkCable, Length=10, Version=1.0.0.3]]
  DriveConfiguration:
    McTypeID = LLMConfig
  DriveConfiguration/Segment:
    Shape = CIRCULAR_TO_STRAIGHT105
    SegmentReference = gSegB10
    SegmentSectorDirection = Positive
    ElongationCompensation = UseAssemblySetting
    StopReaction = UseAssemblySetting
    SpeedFilter = UseAssemblySetting
SegB11 : 8F1I01.BB4B.xxxx-1 v1.0.0.2  [PLK1 -> SegB12.PLK2 (NodeNumber=11) [Cable Type=PowerlinkCable, Length=10, Version=1.0.0.3]]
  DriveConfiguration:
    McTypeID = LLMConfig
  DriveConfiguration/Segment:
    Shape = CIRCULAR
    SegmentReference = gSegB11
    SegmentSectorDirection = Positive
    ElongationCompensation = UseAssemblySetting
    StopReaction = UseAssemblySetting
    SpeedFilter = UseAssemblySetting
SegB12 : 8F1I01.BB4B.xxxx-1 v1.0.0.2  [PLK1 -> SegB13.PLK2 (NodeNumber=10) [Cable Type=PowerlinkCable, Length=10, Version=1.0.0.3]; PLK2 -> SegB11.PLK1 (NodeNumber=10) [Cable Type=PowerlinkCable, Length=10, Version=1.0.0.3]]
  DriveConfiguration:
    McTypeID = LLMConfig
  DriveConfiguration/Segment:
    Shape = CIRCULAR
    SegmentReference = gSegB12
    SegmentSectorDirection = Positive
    ElongationCompensation = UseAssemblySetting
    StopReaction = UseAssemblySetting
    SpeedFilter = UseAssemblySetting
SegB13 : 8F1I01.BB4B.xxxx-1 v1.0.0.2  [PLK1 -> SegB14.PLK2 (NodeNumber=9) [Cable Type=PowerlinkCable, Length=10, Version=1.0.0.3]; PLK2 -> SegB12.PLK1 (NodeNumber=9) [Cable Type=PowerlinkCable, Length=10, Version=1.0.0.3]]
  DriveConfiguration:
    McTypeID = LLMConfig
  DriveConfiguration/Segment:
    Shape = CIRCULAR
    SegmentReference = gSegB13
    SegmentSectorDirection = Positive
    ElongationCompensation = UseAssemblySetting
    StopReaction = UseAssemblySetting
    SpeedFilter = UseAssemblySetting
SegB14 : 8F1I01.AB2B.xxxx-1 v1.0.0.2  [PLK1 -> SegB15.PLK2 (NodeNumber=8) [Cable Type=PowerlinkCable, Length=10, Version=1.0.0.3]; PLK2 -> SegB13.PLK1 (NodeNumber=8) [Cable Type=PowerlinkCable, Length=10, Version=1.0.0.3]]
  DriveConfiguration:
    McTypeID = LLMConfig
  DriveConfiguration/Segment:
    Shape = STRAIGHT105_TO_CIRCULAR
    SegmentReference = gSegB14
    SegmentSectorDirection = Positive
    ElongationCompensation = UseAssemblySetting
    StopReaction = UseAssemblySetting
    SpeedFilter = UseAssemblySetting
SegB15 : 8F1I01.AB2B.xxxx-1 v1.0.0.2  [PLK1 -> SegB16.PLK2 (NodeNumber=7) [Cable Type=PowerlinkCable, Length=10, Version=1.0.0.3]; PLK2 -> SegB14.PLK1 (NodeNumber=7) [Cable Type=PowerlinkCable, Length=10, Version=1.0.0.3]]
  DriveConfiguration:
    McTypeID = LLMConfig
  DriveConfiguration/Segment:
    Shape = STRAIGHT105_TO_CIRCULAR
    SegmentReference = gSegB15
    SegmentSectorDirection = Positive
    ElongationCompensation = UseAssemblySetting
    StopReaction = UseAssemblySetting
    SpeedFilter = UseAssemblySetting
SegB16 : 8F1I01.BA2B.xxxx-1 v1.0.0.2  [PLK1 -> SegB17.PLK2 (NodeNumber=6) [Cable Type=PowerlinkCable, Length=10, Version=1.0.0.3]; PLK2 -> SegB15.PLK1 (NodeNumber=6) [Cable Type=PowerlinkCable, Length=10, Version=1.0.0.3]]
  DriveConfiguration:
    McTypeID = LLMConfig
  DriveConfiguration/Segment:
    Shape = CIRCULAR_TO_STRAIGHT105
    SegmentReference = gSegB16
    SegmentSectorDirection = Positive
    ElongationCompensation = UseAssemblySetting
    StopReaction = UseAssemblySetting
    SpeedFilter = UseAssemblySetting
SegB17 : 8F1I01.BA2B.xxxx-1 v1.0.0.2  [PLK1 -> SegB18.PLK2 (NodeNumber=5) [Cable Type=PowerlinkCable, Length=10, Version=1.0.0.3]; PLK2 -> SegB16.PLK1 (NodeNumber=5) [Cable Type=PowerlinkCable, Length=10, Version=1.0.0.3]]
  DriveConfiguration:
    McTypeID = LLMConfig
  DriveConfiguration/Segment:
    Shape = CIRCULAR_TO_STRAIGHT105
    SegmentReference = gSegB17
    SegmentSectorDirection = Positive
    ElongationCompensation = UseAssemblySetting
    StopReaction = UseAssemblySetting
    SpeedFilter = UseAssemblySetting
SegB18 : 8F1I01.AB2B.xxxx-1 v1.0.0.2  [PLK1 -> SegB1.PLK2 (NodeNumber=4) [Cable Type=PowerlinkCable, Length=10, Version=1.0.0.3]; PLK2 -> SegB17.PLK1 (NodeNumber=4) [Cable Type=PowerlinkCable, Length=10, Version=1.0.0.3]]
  DriveConfiguration:
    McTypeID = LLMConfig
  DriveConfiguration/Segment:
    Shape = STRAIGHT105_TO_CIRCULAR
    SegmentReference = gSegB18
    SegmentSectorDirection = Positive
    ElongationCompensation = UseAssemblySetting
    StopReaction = UseAssemblySetting
    SpeedFilter = UseAssemblySetting
SegB2 : 8F1I01.BB4B.xxxx-1 v1.0.0.2  [PLK1 -> SegB3.PLK2 (NodeNumber=13) [Cable Type=PowerlinkCable, Length=10, Version=1.0.0.3]; PLK2 -> SegB1.PLK1 (NodeNumber=13) [Cable Type=PowerlinkCable, Length=10, Version=1.0.0.3]]
  DriveConfiguration:
    McTypeID = LLMConfig
  DriveConfiguration/Segment:
    Shape = CIRCULAR
    SegmentReference = gSegB2
    SegmentSectorDirection = Positive
    ElongationCompensation = UseAssemblySetting
    StopReaction = UseAssemblySetting
    SpeedFilter = UseAssemblySetting
SegB3 : 8F1I01.BB4B.xxxx-1 v1.0.0.2  [PLK1 -> SegB4.PLK2 (NodeNumber=14) [Cable Type=PowerlinkCable, Length=10, Version=1.0.0.3]; PLK2 -> SegB2.PLK1 (NodeNumber=14) [Cable Type=PowerlinkCable, Length=10, Version=1.0.0.3]]
  DriveConfiguration:
    McTypeID = LLMConfig
  DriveConfiguration/Segment:
    Shape = CIRCULAR
    SegmentReference = gSegB3
    SegmentSectorDirection = Positive
    ElongationCompensation = UseAssemblySetting
    StopReaction = UseAssemblySetting
    SpeedFilter = UseAssemblySetting
SegB4 : 8F1I01.BB4B.xxxx-1 v1.0.0.2  [PLK1 -> SegB5.PLK2 (NodeNumber=15) [Cable Type=PowerlinkCable, Length=10, Version=1.0.0.3]; PLK2 -> SegB3.PLK1 (NodeNumber=15) [Cable Type=PowerlinkCable, Length=10, Version=1.0.0.3]]
  DriveConfiguration:
    McTypeID = LLMConfig
  DriveConfiguration/Segment:
    Shape = CIRCULAR
    SegmentReference = gSegB4
    SegmentSectorDirection = Positive
    ElongationCompensation = UseAssemblySetting
    StopReaction = UseAssemblySetting
    SpeedFilter = UseAssemblySetting
SegB5 : 8F1I01.AB2B.xxxx-1 v1.0.0.2  [PLK1 -> SegB6.PLK2 (NodeNumber=16) [Cable Type=PowerlinkCable, Length=10, Version=1.0.0.3]; PLK2 -> SegB4.PLK1 (NodeNumber=16) [Cable Type=PowerlinkCable, Length=10, Version=1.0.0.3]]
  DriveConfiguration:
    McTypeID = LLMConfig
  DriveConfiguration/Segment:
    Shape = STRAIGHT105_TO_CIRCULAR
    SegmentReference = gSegB5
    SegmentSectorDirection = Positive
    ElongationCompensation = UseAssemblySetting
    StopReaction = UseAssemblySetting
    SpeedFilter = UseAssemblySetting
SegB6 : 8F1I01.AB2B.xxxx-1 v1.0.0.2  [PLK1 -> SegB7.PLK2 (NodeNumber=17) [Cable Type=PowerlinkCable, Length=10, Version=1.0.0.3]; PLK2 -> SegB5.PLK1 (NodeNumber=17) [Cable Type=PowerlinkCable, Length=10, Version=1.0.0.3]]
  DriveConfiguration:
    McTypeID = LLMConfig
  DriveConfiguration/Segment:
    Shape = STRAIGHT105_TO_CIRCULAR
    SegmentReference = gSegB6
    SegmentSectorDirection = Positive
    ElongationCompensation = UseAssemblySetting
    StopReaction = UseAssemblySetting
    SpeedFilter = UseAssemblySetting
SegB7 : 8F1I01.BA2B.xxxx-1 v1.0.0.2  [PLK1 -> SegB8.PLK2 (NodeNumber=18) [Cable Type=PowerlinkCable, Length=10, Version=1.0.0.3]; PLK2 -> SegB6.PLK1 (NodeNumber=18) [Cable Type=PowerlinkCable, Length=10, Version=1.0.0.3]]
  DriveConfiguration:
    McTypeID = LLMConfig
  DriveConfiguration/Segment:
    Shape = CIRCULAR_TO_STRAIGHT105
    SegmentReference = gSegB7
    SegmentSectorDirection = Positive
    ElongationCompensation = UseAssemblySetting
    StopReaction = UseAssemblySetting
    SpeedFilter = UseAssemblySetting
SegB8 : 8F1I01.BA2B.xxxx-1 v1.0.0.2  [PLK1 -> SegB9.PLK2 (NodeNumber=20) [Cable Type=PowerlinkCable, Length=10, Version=1.0.0.3]; PLK2 -> SegB7.PLK1 (NodeNumber=20) [Cable Type=PowerlinkCable, Length=10, Version=1.0.0.3]]
  DriveConfiguration:
    McTypeID = LLMConfig
  DriveConfiguration/Segment:
    Shape = CIRCULAR_TO_STRAIGHT105
    SegmentReference = gSegB8
    SegmentSectorDirection = Positive
    ElongationCompensation = UseAssemblySetting
    StopReaction = UseAssemblySetting
    SpeedFilter = UseAssemblySetting
SegB9 : 8F1I01.AB2B.xxxx-1 v1.0.0.2  [PLK1 -> SegB10.PLK2 (NodeNumber=19) [Cable Type=PowerlinkCable, Length=10, Version=1.0.0.3]; PLK2 -> SegB8.PLK1 (NodeNumber=19) [Cable Type=PowerlinkCable, Length=10, Version=1.0.0.3]]
  DriveConfiguration:
    McTypeID = LLMConfig
  DriveConfiguration/Segment:
    Shape = STRAIGHT105_TO_CIRCULAR
    SegmentReference = gSegB9
    SegmentSectorDirection = Positive
    ElongationCompensation = UseAssemblySetting
    StopReaction = UseAssemblySetting
    SpeedFilter = UseAssemblySetting
X20BB80 : X20BB80 v1.1.0.0
X20BB81a : X20BB81 v1.1.0.0
  Connector IF1:
    ActivateX2X = 0
X20BC0083 : X20BC0083 v2.14.0.0  [PLK1 -> X20HB2880.ETH1 (NodeNumber=33) [Cable Type=PowerlinkCable, Length=10, Version=1.0.0.3]; SL -> X20BB80.SL1]
  Supervision = off
X20BM11 : X20BM11 v1.1.0.0  [X2X1 -> X20BB80.IF1]
X20BT9400 : X20BT9400 v1.3.0.0  [SS1 -> X20TB12b.SS; SL -> X20BM11.SL1]
  Supervision = off
X20HB2880 : X20HB2880 v1.2.0.0  [ETH1 -> X20BC0083.PLK1 [Cable Type=PowerlinkCable, Length=10, Version=1.0.0.3]; ETH2 -> SegB1.PLK3 [Cable Type=PowerlinkCable, Length=10, Version=1.0.0.3]; SS -> X20BB81a.SS1]
X20HB8880 : X20HB8880 v1.1.0.0  [ETH1 -> 5LS182.6-2.IF1 [Cable Type=PowerlinkCable, Length=10, Version=1.0.0.3]; ETH2 -> SegA1.PLK3 [Cable Type=PowerlinkCable, Length=10, Version=1.0.0.3]; SL -> X20BB81a.SL1]
X20PS9400 : X20PS9400 v1.8.0.0  [SS1 -> X20TB12.SS; PS -> X20BB81a.PS1]
  Supervision = off
X20PS9400a : X20PS9400 v1.8.0.0  [SS1 -> X20TB12a.SS; PS -> X20BB80.PS1]
  Supervision = off
X20TB12 : X20TB12 v1.0.0.0
X20TB12a : X20TB12 v1.0.0.0
X20TB12b : X20TB12 v1.0.0.0
```

### Config.mappmotioncfg - 5PC900_TS17_00/mappMotion/Config.mappmotioncfg
```
Element MappMotionConfiguration (Type=mappmotioncfg)
  Processing:
    ProcessingTaskClass = 1
  SharedAlarms:
    Assembly = MpAlarmX
      mapp.AlarmX.Core.Configuration:
        [3]:
          Code = 100
          Severity = 100
    Segment = MpAlarmX
      mapp.AlarmX.Core.Configuration:
        [3]:
          Code = 1100
          Severity = 100
    Sector = MpAlarmX
    Shuttle = MpAlarmX
      mapp.AlarmX.Core.Configuration:
        [3]:
          Code = 2100
          Severity = 100
```

## Logical view

Binary libraries used (declarations not repeated): operator, runtime, astime, AsIecCon, standard, AsBrStr, AsZip, FileIO, AsHttp, brsystem, DataObj, sys_lib, ArEventLog, AsArSdm, MpAlarmX 5.24.3, MpBase, McAcpTrak 5.22.1, McBase, McAxis 5.22.1, CoTrace, MpServer, AsMem, AsUSB, AsICMP, FileExplorer, TrakLib

### Global.var
```iecst
VAR
	gMachineErrorReset : BOOL;
END_VAR
```

- Project.language (not shown)

### ExplorerVariables.var
```iecst
VAR CONSTANT
	EXPL_DIR_PATH_LENGTH : UINT := 200; (*Maximum length for the complete path *)
	EXPL_LIST_NUM : UINT := 100; (*Maximum number if files and folders that can be listed *)
	EXPL_ITEM_LENGTH : USINT := 50; (*Maximum length for a file or folder name *)
	EXPL_SIZE_LENGTH : USINT := 15; (*Maximum length for a file or folder size*)
	EXPL_UPLOAD_DOWNLOAD_SIZE : UDINT := 5000000; (*Maximum size of memory allocated for uploading and downloading files*)
	EXPL_DEVICE_LIST : ARRAY[0..6] OF STRING[40] := ['Diagnosis','USER','USB_DEVICE1','USB_DEVICE2','USB_DEVICE3','NET_DEVICE','']; (*List of predefined devices *)
END_VAR
VAR
	EXPL_VIEW_FILTER : ARRAY[0..9] OF STRING[5] := ['csv','xml','txt','bmp','jpg',5('')]; (*Files extensions than can be used with the view command*)
	EXPL : expMAIN; (*Explorer main structure*)
END_VAR
```

### Library Logical/Trak/Libraries/TrakDiag (ANSIC, version 2.07.2) - https://github.com/hilch/TrakDiag
Depends on: ArEventLog, astime, DataObj, McAcpTrak, standard, McBase, sys_lib, brsystem, FileIO, AsHttp, AsArSdm

#### TD_LogWrite.cpp
```cpp
/*

https://github.com/hilch/TrakDiag

Helper Library for ACOPOStrak diagnosis

MIT License

Copyright (c) 2022 https://github.com/hilch

Permission is hereby granted, free of charge, to any person obtaining a copy
of this software and associated documentation files (the "Software"), to deal
in the Software without restriction, including without limitation the rights
to use, copy, modify, merge, publish, distribute, sublicense, and/or sell
copies of the Software, and to permit persons to whom the Software is
furnished to do so, subject to the following conditions:

The above copyright notice and this permission notice shall be included in all
copies or substantial portions of the Software.

THE SOFTWARE IS PROVIDED "AS IS", WITHOUT WARRANTY OF ANY KIND, EXPRESS OR
IMPLIED, INCLUDING BUT NOT LIMITED TO THE WARRANTIES OF MERCHANTABILITY,
FITNESS FOR A PARTICULAR PURPOSE AND NONINFRINGEMENT. IN NO EVENT SHALL THE
AUTHORS OR COPYRIGHT HOLDERS BE LIABLE FOR ANY CLAIM, DAMAGES OR OTHER
LIABILITY, WHETHER IN AN ACTION OF CONTRACT, TORT OR OTHERWISE, ARISING FROM,
OUT OF OR IN CONNECTION WITH THE SOFTWARE OR THE USE OR OTHER DEALINGS IN THE
SOFTWARE.
*/

#include <bur/plctypes.h>
#include <cstring>
#include <algorithm>

#ifdef __cplusplus
	extern "C"
	{
#endif
	#include "TrakDiag.h"
#ifdef __cplusplus
	};
#endif

/* Write into Logger */
void TD_LogWrite(struct TD_LogWrite* inst)
{
	if( inst->Execute ){
		switch( inst->step ){
			case 0: /* start */
			inst->Busy = 1;
			inst->StatusID = 0;
			std::memset( &inst->fbLogGetIdent, 0, sizeof(inst->fbLogGetIdent) );
			std::strcpy( (char*) &inst->fbLogGetIdent.Name, inst->Name );
			inst->fbLogGetIdent.Execute = 1;
			ArEventLogGetIdent( &inst->fbLogGetIdent );
			if( inst->fbLogGetIdent.Done ){ /* ArEventLogGetIdent is executed synchronously ! */
				std::memset( &inst->fbLogWrite, 0, sizeof(inst->fbLogWrite) );
				ArEventLogWrite( &inst->fbLogWrite ); /* reset fb */
				inst->fbLogWrite.Ident = inst->fbLogGetIdent.Ident;
				inst->fbLogWrite.EventID = inst->EventID;
				inst->fbLogWrite.OriginRecordID = 0;
				inst->fbLogWrite.AddDataSize = std::min( sizeof(inst->Ascii)-1, 1+std::strlen((char*)&inst->Ascii) );
				inst->fbLogWrite.AddData = (UDINT) &inst->Ascii;
				inst->fbLogWrite.AddDataFormat = arEVENTLOG_ADDFORMAT_TEXT;
				std::strcpy( (char*) &inst->fbLogWrite.ObjectID, (char*) &inst->ObjectID );
				inst->fbLogWrite.TimeStamp = 0;
				inst->fbLogWrite.Execute = 1;

				inst->fbLogGetIdent.Execute = 0; /* reset fb */
				ArEventLogGetIdent( &inst->fbLogGetIdent );

				ArEventLogWrite( &inst->fbLogWrite );
				if( inst->fbLogWrite.Done ){ /* ArEventLogWrite is executed synchronously !  */
					inst->fbLogWrite.Execute = 0; /* reset fb */
					ArEventLogWrite( &inst->fbLogWrite );
					inst->Busy = 0;
					inst->Done = 1;
					inst->step = 100;
				}
				else if( inst->fbLogWrite.Error ){
					inst->StatusID = inst->fbLogWrite.StatusID;
					inst->fbLogWrite.Execute = 0; /* reset fb */
					ArEventLogWrite( &inst->fbLogWrite );
					inst->step = 9001;
				}
			}
			else if (inst->fbLogGetIdent.Error ) {
				if( inst->fbLogGetIdent.StatusID == arEVENTLOG_ERR_LOGBOOK_NOT_FOUND ){
					std::memset( &inst->fbLogCreate, 0, sizeof(inst->fbLogCreate) );
					inst->fbLogCreate.Execute = 1;
					std::strcpy( (char*) inst->fbLogCreate.Name, (char*) inst->Name );
					inst->fbLogCreate.Size = 200 * 1024;
					inst->fbLogCreate.Persistence = arEVENTLOG_PERSISTENCE_PERSIST;
					ArEventLogCreate( &inst->fbLogCreate );
					inst->step = 10;
				}
				else {
					inst->StatusID = inst->fbLogGetIdent.StatusID;
					inst->step = 9000;
				}
				inst->fbLogGetIdent.Execute = 0; /* reset fb */
				ArEventLogGetIdent( &inst->fbLogGetIdent );
			}
			break;

			case 10: /* create a new log */
			if( inst->fbLogCreate.Done ){
				inst->fbLogCreate.Execute = 0;
				ArEventLogCreate( &inst->fbLogCreate );
				inst->step = 0;
			}
			else if( inst->fbLogCreate.Error ){
				inst->StatusID = inst->fbLogCreate.StatusID;
				inst->fbLogCreate.Execute = 0;
				ArEventLogCreate( &inst->fbLogCreate );
				inst->step = 9002;
			}
			else {
				ArEventLogCreate( &inst->fbLogCreate );
			}
			break;

			case 100: /* done */

			break;

			case 9000: /* error */
			case 9001:
			case 9002:
			inst->Busy = 0;
			inst->Error = 1;
			break;

		}
	}
	else {
		inst->step = 0;
		inst->Error = 0;
		inst->Busy = 0;
		inst->Done = 0;
	}
}
```

#### TD_LogWatchBOOL.cpp
```cpp
/*

https://github.com/hilch/TrakDiag

Helper Library for ACOPOStrak diagnosis

MIT License

Copyright (c) 2022 https://github.com/hilch

Permission is hereby granted, free of charge, to any person obtaining a copy
of this software and associated documentation files (the "Software"), to deal
in the Software without restriction, including without limitation the rights
to use, copy, modify, merge, publish, distribute, sublicense, and/or sell
copies of the Software, and to permit persons to whom the Software is
furnished to do so, subject to the following conditions:

The above copyright notice and this permission notice shall be included in all
copies or substantial portions of the Software.

THE SOFTWARE IS PROVIDED "AS IS", WITHOUT WARRANTY OF ANY KIND, EXPRESS OR
IMPLIED, INCLUDING BUT NOT LIMITED TO THE WARRANTIES OF MERCHANTABILITY,
FITNESS FOR A PARTICULAR PURPOSE AND NONINFRINGEMENT. IN NO EVENT SHALL THE
AUTHORS OR COPYRIGHT HOLDERS BE LIABLE FOR ANY CLAIM, DAMAGES OR OTHER
LIABILITY, WHETHER IN AN ACTION OF CONTRACT, TORT OR OTHERWISE, ARISING FROM,
OUT OF OR IN CONNECTION WITH THE SOFTWARE OR THE USE OR OTHER DEALINGS IN THE
SOFTWARE.
*/

#include <bur/plctypes.h>
#include <cstring>
#include <cstdio>

#ifdef __cplusplus
	extern "C"
	{
#endif
	#include "TrakDiag.h"
#ifdef __cplusplus
	};
#endif
/* Write status of BOOL variable into log */
void TD_LogWatchBOOL(struct TD_LogWatchBOOL* inst)
{
	if( inst->Enable ){
		switch( inst->step ){
			case 0: /* startup */
			inst->Busy = 1;
			std::memset( &inst->fbLogWrite, 0, sizeof(inst->fbLogWrite) );
			std::strcpy( (char*) inst->fbLogWrite.Name, (char*) inst->LogName );
			inst->signalOld = !inst->Signal;
			inst->step = 10;
			break;

			case 10: /* check signal */
			inst->Valid = 1;
			if( inst->Signal != inst->signalOld){
				inst->signalOld = inst->Signal;
				std::strcpy( (char*) inst->fbLogWrite.ObjectID, (char*) inst->SignalName );
				std::strcpy( (char*) inst->fbLogWrite.Ascii, inst->Signal ? "TRUE" : "FALSE" );
				inst->fbLogWrite.EventID = inst->EventID;
				inst->fbLogWrite.Execute = 1;
				inst->Busy = 1;
				TD_LogWrite( &inst->fbLogWrite );
				if( inst->fbLogWrite.Done ){
					inst->Busy = 0;
					inst->fbLogWrite.Execute = 0;
					TD_LogWrite( &inst->fbLogWrite );
				}
				else if( inst->fbLogWrite.Error ){
					inst->Busy = 0;
					inst->StatusID = inst->fbLogWrite.StatusID;
					inst->fbLogWrite.Execute = 0;
					TD_LogWrite( &inst->fbLogWrite );
					inst->step = 9999;
				}
			}
			break;

			case 9999: /* error */
			inst->Valid = 0;
			inst->Busy = 0;
			inst->Error = 1;
			break;

		}
	}
	else {
		inst->Busy = 0;
		inst->Valid = 0;
		inst->StatusID = 0;
		inst->Error = 0;
		inst->step = 0;
	}
}
```

#### TD_LogWatchDINT.cpp
```cpp
/*

https://github.com/hilch/TrakDiag

Helper Library for ACOPOStrak diagnosis

MIT License

Copyright (c) 2022 https://github.com/hilch

Permission is hereby granted, free of charge, to any person obtaining a copy
of this software and associated documentation files (the "Software"), to deal
in the Software without restriction, including without limitation the rights
to use, copy, modify, merge, publish, distribute, sublicense, and/or sell
copies of the Software, and to permit persons to whom the Software is
furnished to do so, subject to the following conditions:

The above copyright notice and this permission notice shall be included in all
copies or substantial portions of the Software.

THE SOFTWARE IS PROVIDED "AS IS", WITHOUT WARRANTY OF ANY KIND, EXPRESS OR
IMPLIED, INCLUDING BUT NOT LIMITED TO THE WARRANTIES OF MERCHANTABILITY,
FITNESS FOR A PARTICULAR PURPOSE AND NONINFRINGEMENT. IN NO EVENT SHALL THE
AUTHORS OR COPYRIGHT HOLDERS BE LIABLE FOR ANY CLAIM, DAMAGES OR OTHER
LIABILITY, WHETHER IN AN ACTION OF CONTRACT, TORT OR OTHERWISE, ARISING FROM,
OUT OF OR IN CONNECTION WITH THE SOFTWARE OR THE USE OR OTHER DEALINGS IN THE
SOFTWARE.
*/

#include <bur/plctypes.h>
#include <cstring>
#include <cstdio>

#ifdef __cplusplus
	extern "C"
	{
#endif
	#include "TrakDiag.h"
#ifdef __cplusplus
	};
#endif
/* Write status of DINT variable into log */
void TD_LogWatchDINT(struct TD_LogWatchDINT* inst)
{
	if( inst->Enable ){
		switch( inst->step ){
			case 0: /* startup */
			inst->Busy = 1;
			std::memset( &inst->fbLogWrite, 0, sizeof(inst->fbLogWrite) );
			std::strcpy( (char*) inst->fbLogWrite.Name, (char*) inst->LogName );
			inst->signalOld = !inst->Signal;
			inst->step = 10;
			break;

			case 10: /* check signal */
			inst->Valid = 1;
			if( inst->Signal != inst->signalOld){
				inst->signalOld = inst->Signal;
				std::strcpy( (char*) inst->fbLogWrite.ObjectID, (char*) inst->SignalName );
				std::sprintf( (char*) inst->fbLogWrite.Ascii, "%ld (0x%x)", inst->Signal, (unsigned int) inst->Signal );
				inst->fbLogWrite.EventID = inst->EventID;
				inst->fbLogWrite.Execute = 1;
				inst->Busy = 1;
				TD_LogWrite( &inst->fbLogWrite );
				if( inst->fbLogWrite.Done ){
					inst->Busy = 0;
					inst->fbLogWrite.Execute = 0; /* reset fb */
					TD_LogWrite( &inst->fbLogWrite );
				}
				else if( inst->fbLogWrite.Error ){
					inst->Busy = 0;
					inst->StatusID = inst->fbLogWrite.StatusID;
					inst->fbLogWrite.Execute = 0;
					TD_LogWrite( &inst->fbLogWrite );
					inst->step = 9999;
				}
			}
			break;

			case 9999: /* error */
			inst->Valid = 0;
			inst->Busy = 0;
			inst->Error = 1;
			break;

		}
	}
	else {
		inst->Busy = 0;
		inst->Valid = 0;
		inst->StatusID = 0;
		inst->Error = 0;
		inst->step = 0;
	}
}
```

#### TD_LogWatchSTRING.cpp
```cpp
/*

https://github.com/hilch/TrakDiag

Helper Library for ACOPOStrak diagnosis

MIT License

Copyright (c) 2022 https://github.com/hilch

Permission is hereby granted, free of charge, to any person obtaining a copy
of this software and associated documentation files (the "Software"), to deal
in the Software without restriction, including without limitation the rights
to use, copy, modify, merge, publish, distribute, sublicense, and/or sell
copies of the Software, and to permit persons to whom the Software is
furnished to do so, subject to the following conditions:

The above copyright notice and this permission notice shall be included in all
copies or substantial portions of the Software.

THE SOFTWARE IS PROVIDED "AS IS", WITHOUT WARRANTY OF ANY KIND, EXPRESS OR
IMPLIED, INCLUDING BUT NOT LIMITED TO THE WARRANTIES OF MERCHANTABILITY,
FITNESS FOR A PARTICULAR PURPOSE AND NONINFRINGEMENT. IN NO EVENT SHALL THE
AUTHORS OR COPYRIGHT HOLDERS BE LIABLE FOR ANY CLAIM, DAMAGES OR OTHER
LIABILITY, WHETHER IN AN ACTION OF CONTRACT, TORT OR OTHERWISE, ARISING FROM,
OUT OF OR IN CONNECTION WITH THE SOFTWARE OR THE USE OR OTHER DEALINGS IN THE
SOFTWARE.
*/

#include <bur/plctypes.h>
#include <cstring>
#include <cstdio>

#ifdef __cplusplus
	extern "C"
	{
#endif
	#include "TrakDiag.h"
#ifdef __cplusplus
	};
#endif
/* Write contents of STRING variable into log */
void TD_LogWatchSTRING(struct TD_LogWatchSTRING* inst)
{
	if( inst->Enable ){
		switch( inst->step ){
			case 0: /* startup */
			inst->Busy = 1;
			std::memset( &inst->fbLogWrite, 0, sizeof(inst->fbLogWrite) );
			std::strcpy( (char*) inst->fbLogWrite.Name, (char*) inst->LogName );
			std::strcpy( (char*) inst->signalOld , "!" );
			std::strcat( (char*) inst->signalOld , (char*) inst->Signal );
			inst->step = 10;
			break;

			case 10: /* check signal */
			inst->Valid = 1;
			if( std::strcmp( (char*) inst->Signal, (char*) inst->signalOld ) ){
				std::strcpy( (char*) inst->signalOld ,(char*) inst->Signal );
				std::strcpy( (char*) inst->fbLogWrite.ObjectID, (char*) inst->SignalName );
				std::strcpy( (char*) inst->fbLogWrite.Ascii, (char*) inst->Signal );
				inst->fbLogWrite.EventID = inst->EventID;
				inst->fbLogWrite.Execute = 1;
				inst->Busy = 1;
				TD_LogWrite( &inst->fbLogWrite );
				if( inst->fbLogWrite.Done ){
					inst->Busy = 0;
					inst->fbLogWrite.Execute = 0;
					TD_LogWrite( &inst->fbLogWrite );
					inst->step = 10;
				}
				else if( inst->fbLogWrite.Error ){
					inst->Busy = 0;
					inst->StatusID = inst->fbLogWrite.StatusID;
					inst->fbLogWrite.Execute = 0;
					TD_LogWrite( &inst->fbLogWrite );
					inst->step = 9999;
				}
			}
			break;

			case 9999: /* error */
			inst->Valid = 0;
			inst->Busy = 0;
			inst->Error = 1;
			break;

		}
	}
	else {
		inst->Busy = 0;
		inst->Valid = 0;
		inst->StatusID = 0;
		inst->Error = 0;
		inst->step = 0;
	}
}
```

#### TD_LogWatch8Flags.cpp
```cpp
/*

https://github.com/hilch/TrakDiag

Helper Library for ACOPOStrak diagnosis

MIT License

Copyright (c) 2022 https://github.com/hilch

Permission is hereby granted, free of charge, to any person obtaining a copy
of this software and associated documentation files (the "Software"), to deal
in the Software without restriction, including without limitation the rights
to use, copy, modify, merge, publish, distribute, sublicense, and/or sell
copies of the Software, and to permit persons to whom the Software is
furnished to do so, subject to the following conditions:

The above copyright notice and this permission notice shall be included in all
copies or substantial portions of the Software.

THE SOFTWARE IS PROVIDED "AS IS", WITHOUT WARRANTY OF ANY KIND, EXPRESS OR
IMPLIED, INCLUDING BUT NOT LIMITED TO THE WARRANTIES OF MERCHANTABILITY,
FITNESS FOR A PARTICULAR PURPOSE AND NONINFRINGEMENT. IN NO EVENT SHALL THE
AUTHORS OR COPYRIGHT HOLDERS BE LIABLE FOR ANY CLAIM, DAMAGES OR OTHER
LIABILITY, WHETHER IN AN ACTION OF CONTRACT, TORT OR OTHERWISE, ARISING FROM,
OUT OF OR IN CONNECTION WITH THE SOFTWARE OR THE USE OR OTHER DEALINGS IN THE
SOFTWARE.
*/

#include <bur/plctypes.h>
#include <cstring>
#include <cstdio>
#include <cctype>
#include <algorithm>

#ifdef __cplusplus
	extern "C"
	{
#endif
	#include "TrakDiag.h"
#ifdef __cplusplus
	};
#endif
/* Write status of 8 flags variable into log */
void TD_LogWatch8Flags(struct TD_LogWatch8Flags* inst)
{
	if( inst->Enable ){
		switch( inst->step ){
			case 0: /* startup */
			inst->Busy = 1;
			std::memset( &inst->fbLogWrite, 0, sizeof(inst->fbLogWrite) );
			std::strcpy( (char*) inst->fbLogWrite.Name, (char*) inst->LogName );
			inst->signalOld = !inst->Signal;
			inst->step = 10;
			break;

			case 10: /* check signal */
			inst->Valid = 1;
			if( inst->Signal != inst->signalOld){

				std::strcpy( (char*) inst->fbLogWrite.ObjectID, (char*) inst->SignalName );
				std::strcpy( (char*) inst->fbLogWrite.Ascii, "" );
				for( int n = 7; n>=0 ; --n ){
					if( inst->Flag[n][0] ){  /* flag used ? */
						char f[sizeof(inst->Flag[0])];
						bool bit = !!(inst->Signal & 1<<n);
						bool bitOld = !!(inst->signalOld & 1<<n);

						std::memset( (void*) &f, 0, sizeof(f) );
						/* use upper case letters for TRUE and lower case for FALSE */
						if( bit ) {
							std::transform( &inst->Flag[n][0], &inst->Flag[n][8], f, std::toupper );
						}
						else {
							std::transform( &inst->Flag[n][0], &inst->Flag[n][8], f, std::tolower );
						}
						/* add a star '*' as prefix if flag was changed */
						if( bit != bitOld ){
							std::strcat( (char*) inst->fbLogWrite.Ascii, "*" );
						}
						else {
							std::strcat( (char*) inst->fbLogWrite.Ascii, " " );
						}
						std::strcat( (char*) inst->fbLogWrite.Ascii, f );
						std::strcat( (char*) inst->fbLogWrite.Ascii, " " );
					}
				}
				inst->signalOld = inst->Signal;
				inst->fbLogWrite.EventID = inst->EventID;
				inst->fbLogWrite.Execute = 1;
				inst->Busy = 1;
				TD_LogWrite( &inst->fbLogWrite );
				if( inst->fbLogWrite.Done ){
					inst->Busy = 0;
					inst->fbLogWrite.Execute = 0;
					TD_LogWrite( &inst->fbLogWrite );
					inst->step = 10;
				}
				else if( inst->fbLogWrite.Error ){
					inst->Busy = 0;
					inst->StatusID = inst->fbLogWrite.StatusID;
					inst->fbLogWrite.Execute = 0;
					TD_LogWrite( &inst->fbLogWrite );
					inst->step = 9999;
				}
			}
			break;

			case 9999: /* error */
			inst->Valid = 0;
			inst->Busy = 0;
			inst->Error = 1;
			break;

		}
	}
	else {
		inst->Busy = 0;
		inst->Valid = 0;
		inst->StatusID = 0;
		inst->Error = 0;
		inst->step = 0;
	}
}
```

#### TD_CrashReport.cpp
```cpp
/*

https://github.com/hilch/TrakDiag

Helper Library for ACOPOStrak diagnosis

MIT License

Copyright (c) 2022 https://github.com/hilch

Permission is hereby granted, free of charge, to any person obtaining a copy
of this software and associated documentation files (the "Software"), to deal
in the Software without restriction, including without limitation the rights
to use, copy, modify, merge, publish, distribute, sublicense, and/or sell
copies of the Software, and to permit persons to whom the Software is
furnished to do so, subject to the following conditions:

The above copyright notice and this permission notice shall be included in all
copies or substantial portions of the Software.

THE SOFTWARE IS PROVIDED "AS IS", WITHOUT WARRANTY OF ANY KIND, EXPRESS OR
IMPLIED, INCLUDING BUT NOT LIMITED TO THE WARRANTIES OF MERCHANTABILITY,
FITNESS FOR A PARTICULAR PURPOSE AND NONINFRINGEMENT. IN NO EVENT SHALL THE
AUTHORS OR COPYRIGHT HOLDERS BE LIABLE FOR ANY CLAIM, DAMAGES OR OTHER
LIABILITY, WHETHER IN AN ACTION OF CONTRACT, TORT OR OTHERWISE, ARISING FROM,
OUT OF OR IN CONNECTION WITH THE SOFTWARE OR THE USE OR OTHER DEALINGS IN THE
SOFTWARE.
*/

#ifndef _REPLACE_CONST
#define _REPLACE_CONST
#endif

#include <bur/plctypes.h>
#include <cstring>
#include <cstdio>
#include <ctime>
#include <algorithm>

#ifdef __cplusplus
	extern "C"
	{
#endif
	#include "TrakDiag.h"
#ifdef __cplusplus
	};
#endif

/* check if we want this entry */

bool isValidEntry( struct TD_CrashReport* inst ){
			bool validSeverity = (inst->fbReadEntry.Entry.Severity >= inst->thrSeverity);

			if( strlen( inst->objectStartsWith1 ) )
				if( std::strstr( inst->fbReadEntry.Entry.ObjectID, inst->objectStartsWith1) )
					return validSeverity;

			if( strlen( inst->objectStartsWith2 ) )
				if( std::strstr( inst->fbReadEntry.Entry.ObjectID, inst->objectStartsWith2) )
					return validSeverity;

			return false;

}

#define W_COMMAND 0
#define GET_IDENT 10
#define W_ENTRIES_WRITTEN 20
#define READ_LATEST_RECORD 30
#define READ_PREVIOUS_ID 40
#define COPY_ENTRY 50
#define READY 100
#define ERROR_GET_IDENT 9001
#define ERROR_GET_PREVIOUS_RECORD_ID 9002
#define ERROR_GET_LATEST_RECORD_ID 9003
#define ERROR_READ_FIRST_ENTRY 9004
#define ERROR_READ_ENTRY 9005

/* read motion logger cyclically */
void TD_CrashReport(struct TD_CrashReport* inst) {

	if( !inst->Execute ){
		inst->step = W_COMMAND;
	}

	for(;;) /* use 'continue' instead of 'break' to save one cycle */
	{
		switch( inst->step ) {

			case W_COMMAND:  /* Execute := FALSE */
			inst->Busy = 0;
			inst->Done = 0;
			inst->Error = 0;
			inst->StatusID = 0;

			if( inst->Execute && inst->pLoggerEntries && (inst->SizeLoggerEntries >= sizeof(TD_LoggerEntryType) ) ) {

				std::memset( (void*) &inst->fbGetIdent, 0, sizeof(inst->fbGetIdent));
				ArEventLogGetIdent( &inst->fbGetIdent );	/* reset fb */

				std::memset( (void*) &inst->fbGetLatestRecordID, 0, sizeof(inst->fbGetLatestRecordID));
				ArEventLogGetLatestRecordID( &inst->fbGetLatestRecordID ); /* reset fb */

				std::memset( (void*) &inst->fbGetPreviousRecordID, 0, sizeof(inst->fbGetPreviousRecordID));
				ArEventLogGetPreviousRecordID( &inst->fbGetPreviousRecordID ); /* reset fb */

				std::memset( (void*) &inst->fbReadEntry, 0, sizeof(inst->fbReadEntry));
				TD_LoggerReadEntry( &inst->fbReadEntry ); /* reset fb */

				std::memset( (void*) &inst->tonDelayRead, 0, sizeof(inst->tonDelayRead));
				TON( &inst->tonDelayRead ); /* reset fb */

				inst->MaxEntries = inst->SizeLoggerEntries / sizeof(TD_LoggerEntryType);
				inst->NbrOfEntries = 0;
				inst->counterEntries = 0;
				std::memset( reinterpret_cast<TD_LoggerEntryType*>(inst->pLoggerEntries),0, inst->SizeLoggerEntries );  /* clear logger entries */

				inst->fbDTGetTime.enable = 1;
				DTGetTime( &inst->fbDTGetTime );
				if( inst->observationPeriod == 0 )
					inst->observationPeriod = 3000; /* 3 seconds */
				inst->eventTimeMinimum = inst->fbDTGetTime.DT1 - inst->observationPeriod/1000;

				inst->Busy = 1;
				inst->index = 0;
				inst->fbGetIdent.Execute = 1;
				std::strcpy( (char*) &inst->fbGetIdent.Name, "$motion" );
				ArEventLogGetIdent( &inst->fbGetIdent );
				inst->step = GET_IDENT;

			}
			break;

			case GET_IDENT: /* get ident of logger module */
			if( inst->fbGetIdent.Done ) {
				inst->fbGetPreviousRecordID.Ident = inst->fbGetIdent.Ident;
				inst->fbReadEntry.Ident = inst->fbGetIdent.Ident;
				inst->fbGetLatestRecordID.Ident = inst->fbGetIdent.Ident;
				inst->tonDelayRead.PT = 1000;
				inst->tonDelayRead.IN = 1;
				inst->step = W_ENTRIES_WRITTEN;
			}
			else if( inst->fbGetIdent.Error ) { /* error getting logger ident for module copy */
				inst->StatusID = inst->fbGetIdent.StatusID;
				inst->step = ERROR_GET_IDENT;
			}
			else { /* busy */
				ArEventLogGetIdent( &inst->fbGetIdent );
			}
			break;

			case W_ENTRIES_WRITTEN: /* wait until entries have been written to logger */
			TON( &inst->tonDelayRead );
			if( inst->tonDelayRead.Q ){
				inst->fbGetLatestRecordID.Execute = 1;
				ArEventLogGetLatestRecordID( &inst->fbGetLatestRecordID );
				inst->step = READ_LATEST_RECORD;
			}
			break;

			case READ_LATEST_RECORD:  /* read lates record id */
			if( inst->fbGetLatestRecordID.Done )
			{
				inst->counterEntries++;
				inst->fbReadEntry.RecordID = inst->fbGetLatestRecordID.RecordID;
				inst->fbReadEntry.Execute = 1;
				TD_LoggerReadEntry( &inst->fbReadEntry );
				inst->NbrOfEntries = 0;
				inst->fbGetLatestRecordID.Execute = 0;
				ArEventLogGetLatestRecordID( &inst->fbGetLatestRecordID );
				inst->step = COPY_ENTRY;
				continue;
			}
			else if( inst->fbGetLatestRecordID.Error ){
				inst->StatusID = inst->fbGetLatestRecordID.StatusID;
				inst->step = ERROR_GET_LATEST_RECORD_ID;
			}
			else {
				ArEventLogGetLatestRecordID( &inst->fbGetLatestRecordID );
			}
			break;

			case READ_PREVIOUS_ID: /* read previous entry */
			if( inst->index < inst->MaxEntries ) {  /* do we have enough space in entries array ? */
				if( inst->fbGetPreviousRecordID.Done ) {
					inst->counterEntries++;
					inst->fbReadEntry.RecordID = inst->fbGetPreviousRecordID.PrevRecordID;
					inst->fbReadEntry.Execute = 1;
					TD_LoggerReadEntry( &inst->fbReadEntry );
					inst->fbGetPreviousRecordID.Execute = 0;
					ArEventLogGetPreviousRecordID( &inst->fbGetPreviousRecordID );
					inst->step = COPY_ENTRY;
					continue;
				}
				else if( inst->fbGetPreviousRecordID.Error ) {
					if( inst->fbGetPreviousRecordID.StatusID == arEVENTLOG_ERR_RECORDID_INVALID ) {  /* end of logger ? */
						inst->step = READY;
						inst->fbGetPreviousRecordID.Execute = 0;
						ArEventLogGetPreviousRecordID( &inst->fbGetPreviousRecordID );
					}
					else {
						inst->StatusID = inst->fbGetPreviousRecordID.StatusID;
						inst->step = ERROR_GET_PREVIOUS_RECORD_ID;
					}
				}
			}
			else { /* maximum number of allowed entries reached */
				inst->step = READY;
				inst->fbGetPreviousRecordID.Execute = 0;
				ArEventLogGetPreviousRecordID( &inst->fbGetPreviousRecordID );
			}
			break;

			case COPY_ENTRY: /* read all data from entry */
			if( inst->fbReadEntry.Done ) {
				if( inst->fbReadEntry.Entry.LocalTime < inst->eventTimeMinimum ){ /* is message out of time scope ? */
					inst->fbGetPreviousRecordID.Execute = 0;
					ArEventLogGetPreviousRecordID( &inst->fbGetPreviousRecordID );
					inst->step = READY;
				}
				else {
					if( isValidEntry(inst) ){ /* does entry fit to the filter ? */
						TD_LoggerEntryType* entry = reinterpret_cast<TD_LoggerEntryType*>(inst->pLoggerEntries);
						if( inst->index > 0 ){ /* only valid if we have two or more entries already */
							for( int i = (inst->MaxEntries-1); i > inst->index; --i ){  /* shift list and remove oldest entry */
								entry[i] = entry[i-1];
							}
						}
						entry[inst->index] = inst->fbReadEntry.Entry;
						++inst->index;
						if( ++inst->NbrOfEntries > inst->MaxEntries )
							inst->NbrOfEntries = inst->MaxEntries;
					}
					else  { /* entry does not fit to filter */
						inst->index = inst->index;
					}
					inst->fbGetPreviousRecordID.RecordID = inst->fbReadEntry.RecordID; /* prepare for next call */
					inst->fbGetPreviousRecordID.Execute = 1;
					ArEventLogGetPreviousRecordID( &inst->fbGetPreviousRecordID );
					inst->fbReadEntry.Execute = 0;
					inst->step = READ_PREVIOUS_ID;
				}
			}
			else if( inst->fbReadEntry.Error ) {
				inst->StatusID = inst->fbReadEntry.StatusID;
				inst->step = ERROR_READ_ENTRY;
			}
			TD_LoggerReadEntry( &inst->fbReadEntry );
			break;

			case READY: /* done */
			inst->Error = 0;
			inst->Busy = 0;
			inst->Done = 1;
			break;

			case ERROR_GET_IDENT: /* internal errors */
			case ERROR_GET_PREVIOUS_RECORD_ID:
			case ERROR_GET_LATEST_RECORD_ID:
			case ERROR_READ_ENTRY:
			case ERROR_READ_FIRST_ENTRY:

			inst->Error = 1;
			inst->Busy = 0;
			inst->Done = 0;
			break;

		} /* end of switch() */
		break; /* exit for */
	} /* end of for() */
}
```

#### TD_SegCommandError.cpp
```cpp
/*

https://github.com/hilch/TrakDiag

Helper Library for ACOPOStrak diagnosis

MIT License

Copyright (c) 2022 https://github.com/hilch

Permission is hereby granted, free of charge, to any person obtaining a copy
of this software and associated documentation files (the "Software"), to deal
in the Software without restriction, including without limitation the rights
to use, copy, modify, merge, publish, distribute, sublicense, and/or sell
copies of the Software, and to permit persons to whom the Software is
furnished to do so, subject to the following conditions:

The above copyright notice and this permission notice shall be included in all
copies or substantial portions of the Software.

THE SOFTWARE IS PROVIDED "AS IS", WITHOUT WARRANTY OF ANY KIND, EXPRESS OR
IMPLIED, INCLUDING BUT NOT LIMITED TO THE WARRANTIES OF MERCHANTABILITY,
FITNESS FOR A PARTICULAR PURPOSE AND NONINFRINGEMENT. IN NO EVENT SHALL THE
AUTHORS OR COPYRIGHT HOLDERS BE LIABLE FOR ANY CLAIM, DAMAGES OR OTHER
LIABILITY, WHETHER IN AN ACTION OF CONTRACT, TORT OR OTHERWISE, ARISING FROM,
OUT OF OR IN CONNECTION WITH THE SOFTWARE OR THE USE OR OTHER DEALINGS IN THE
SOFTWARE.
*/

#include <bur/plctypes.h>
#include <cstring>

#ifdef __cplusplus
	extern "C"
	{
#endif
	#include "TrakDiag.h"
#ifdef __cplusplus
	};
#endif

/* Simulate Segment Error */
void TD_SegCommandError(struct TD_SegCommandError* inst)
{

	if( !inst->Execute )
		inst->step = 0;

	switch( inst->step ){
		case 0:
		inst->Busy = 0;
		inst->Done = 0;
		inst->Error = 0;
		inst->StatusID = 0;
		if( inst->Execute ){
			inst->Busy = 1;
			std::memset( &inst->fbSegPowerOn, 0, sizeof(inst->fbSegPowerOn) );
			MC_BR_SegPowerOn_AcpTrak( &inst->fbSegPowerOn ); /* reset fb */

			std::memset( &inst->fbSegCommandError, 0, sizeof(inst->fbSegCommandError) );
			MC_BR_SegCommandError_AcpTrak( &inst->fbSegCommandError ); /* reset fb */
			inst->fbSegCommandError.Segment = inst->Segment;
			switch( inst->Type ){
				case TD_SEGERRCMD_SEGMENT: inst->fbSegCommandError.Command = mcERROR_CMD; break;
				case TD_SEGERRCMD_CHANNEL: inst->fbSegCommandError.Command = mcERROR_CHANNEL_CMD; break;
				case TD_SEGERRCMD_ENCODER: inst->fbSegCommandError.Command = mcERROR_ENCODER_CMD; break;
			}
			inst->fbSegCommandError.Execute = 1;
			MC_BR_SegCommandError_AcpTrak( &inst->fbSegCommandError );
			inst->step = 10;
		}
		break;

		case 10: /* send error command to segment */
		if( inst->fbSegCommandError.Done ){
			if( inst->fbSegCommandError.Command == mcERROR_CMD ){ /* mcERROR_CMD requires a subsequent command */
				inst->fbSegPowerOn.Segment = inst->Segment;
				inst->fbSegPowerOn.Execute = 1;
				MC_BR_SegPowerOn_AcpTrak( &inst->fbSegPowerOn );
				inst->step = 20;
			}
			else {
				inst->step = 100;
			}
		}
		else if( inst->fbSegCommandError.Error ){
			inst->StatusID = inst->fbSegCommandError.ErrorID;
			inst->step = 9001;
		}
		else { /* busy */
			MC_BR_SegCommandError_AcpTrak( &inst->fbSegCommandError );
		}
		break;

		case 20: /* try to power on segment in errorstop (which will fail!) */
		if( inst->fbSegPowerOn.Done || inst->fbSegPowerOn.Error ){
			inst->step = 100;
		}
		else {  /* busy */
			MC_BR_SegPowerOn_AcpTrak( &inst->fbSegPowerOn );
		}

		case 100: /* Done */
		inst->Busy = 0;
		inst->Done = 1;
		break;

		case 9001: /* internal errors */
		inst->Busy = 0;
		inst->Error = 1;
		break;

	}
}
```

### Program Logical/Trak/SegCtrl (IEC)

#### Init.st
```iecst
PROGRAM _INIT
	gSegA1;
	gSegA2;
	gSegA3;
	gSegA4;
	gSegA5;
	gSegA6;
	gSegA7;
	gSegA8;
	gSegA9;
	gSegA10;
	gSegA11;
	gSegA12;
	gSegA13;
	gSegA14;

	gSegB1;
	gSegB2;
	gSegB3;
	gSegB4;
	gSegB5;
	gSegB6;
	gSegB7;
	gSegB8;
	gSegB9;
	gSegB10;
	gSegB11;
	gSegB12;
	gSegB13;
	gSegB14;
	gSegB15;
	gSegB16;
	gSegB17;
	gSegB18;

END_PROGRAM
```

Listed in the project but not available here: Logical/NETdevice/NetTypes.typ, Logical/NETdevice/NetVariables.var, Logical/NETdevice/NetDevice, Logical/Trak/Assembly.typ, Logical/Trak/Libraries/TrakDiag/TrakDiagTypes.typ, Logical/Trak/Libraries/TrakDiag/TrakDiagConstants.var, Logical/Trak/Libraries/TrakDiag/TrakDiag.fun, Logical/Trak/Libraries/TrakDiag/TD_ascDT.cpp, Logical/Trak/Libraries/TrakDiag/TD_filenameDT.cpp, Logical/Trak/Libraries/TrakDiag/TD_LoggerReadEntry.cpp, Logical/Trak/Libraries/TrakDiag/TD_Recorder.cpp, Logical/Trak/Libraries/TrakDiag/recorder_html.h, Logical/Trak/Libraries/TrakDiag/TD_Recorder.h, Logical/Trak/Libraries/TrakDiag/TD_WebServices.cpp, Logical/Trak/Libraries/TrakDiag/TD_WebServices.h, Logical/Trak/Libraries/TrakDiag/TD_ShuttleErrorTexts.cpp, Logical/Trak/Libraries/TrakDiag/TD_SegmentsInfo.cpp, Logical/Trak/Libraries/TrakDiag/TD_LimitFileNumber.cpp, Logical/Trak/Libraries/TrakDiag/TD_GetShuttles.cpp, Logical/Trak/Libraries/TrakDiag/TrakWebApi/utils.h, Logical/Trak/Libraries/TrakDiag/TrakWebApi/utils.cpp, Logical/Trak/Libraries/TrakDiag/TrakWebApi/responses.h, Logical/Trak/Libraries/TrakDiag/TrakWebApi/responses.cpp, Logical/Trak/Libraries/TrakDiag/TrakWebApi/index_css.h, Logical/Trak/Libraries/TrakDiag/TrakWebApi/index_js.h, Logical/Trak/Libraries/TrakDiag/TrakWebApi/panzoom_js.h, Logical/Trak/Libraries/TrakDiag/TrakWebApi/index_html.h, Logical/Trak/TrakConstants.var, Logical/Trak/Segments.var, Logical/Trak/TrakInit, Logical/Trak/AssCtrl, Logical/USBdevice/UsbTypes.typ, Logical/USBdevice/UsbVariables.var, Logical/USBdevice/UsbDevice
